KUKA KRL program: MyProgram_260().src

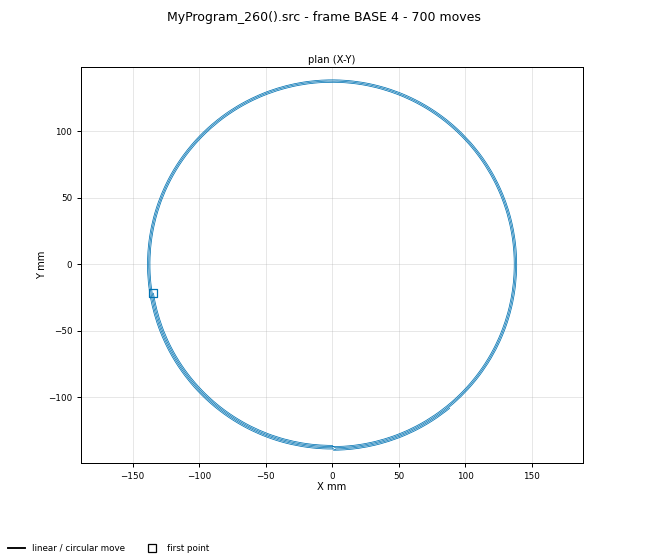
[picture p0: tool path of MyProgram_260().src in frame BASE 4, 700 of 700 moves have a stored position in this frame; points joined in program order, loops and branches not executed]
&ACCESS RVP
&REL 1
&PARAM TEMPLATE = C:\KRC\Roboter\Template\vorgabe
&PARAM EDITMASK = *
DEF MyProgram_260()
; ---- Setting reference (Base) ----
$BASE = BASE_DATA[4]

; --------------------------
; ---- Setting tool (TCP) ----
$TOOL = TOOL_DATA[3]
; --------------------------

$VEL.CP = VEL_APROX_PRINT
Startdeposition()
$VEL.CP = VEL_PRINT
LIN {X -134.3111,Y -21.6727,Z 167,A -169.5198,B 10.842,C 0.1896,E1 10.6856,E2 260.3687} C_DIS
LIN {X -133.7685,Y -24.8029,Z 167,A -167.9998,B 10.842,C 0.1897,E1 10.6864,E2 258.8275} C_DIS
LIN {X -133.0833,Y -28.2434,Z 167,A -166.7087,B 10.8418,C 0.1977,E1 10.6871,E2 257.5607} C_DIS
LIN {X -132.3432,Y -31.5283,Z 167,A -165.3421,B 10.8418,C 0.2028,E1 10.688,E2 256.2017} C_DIS
LIN {X -131.6516,Y -34.3082,Z 167,A -163.8428,B 10.8418,C 0.2002,E1 10.689,E2 254.6673} C_DIS
LIN {X -130.7834,Y -37.4821,Z 167,A -162.445,B 10.8418,C 0.2039,E1 10.6901,E2 253.2692} C_DIS
LIN {X -129.8475,Y -40.6068,Z 167,A -161.0737,B 10.8416,C 0.2077,E1 10.6912,E2 251.8994} C_DIS
LIN {X -128.6869,Y -44.1413,Z 167,A -159.7043,B 10.8415,C 0.216,E1 10.6924,E2 250.5557} C_DIS
LIN {X -127.68,Y -46.9788,Z 167,A -158.313,B 10.8415,C 0.217,E1 10.6937,E2 249.1502} C_DIS
LIN {X -126.4966,Y -50.0788,Z 167,A -156.7273,B 10.8415,C 0.2169,E1 10.6954,E2 247.5422} C_DIS
LIN {X -124.9844,Y -53.7359,Z 167,A -155.1801,B 10.8413,C 0.2238,E1 10.697,E2 246.0111} C_DIS
LIN {X -123.8203,Y -56.3713,Z 167,A -153.9567,B 10.8413,C 0.2268,E1 10.6984,E2 244.7874} C_DIS
LIN {X -122.3652,Y -59.4639,Z 167,A -152.3703,B 10.8413,C 0.2275,E1 10.7004,E2 243.1838} C_DIS
LIN {X -120.7964,Y -62.5886,Z 167,A -151.0422,B 10.8411,C 0.2342,E1 10.702,E2 241.8746} C_DIS
LIN {X -119.2164,Y -65.5493,Z 167,A -149.5746,B 10.8411,C 0.2367,E1 10.704,E2 240.4013} C_DIS
LIN {X -117.5118,Y -68.5582,Z 167,A -147.9691,B 10.8411,C 0.2372,E1 10.7063,E2 238.7782} C_DIS
LIN {X -115.1541,Y -72.4477,Z 167,A -146.0552,B 10.8409,C 0.2419,E1 10.7091,E2 236.8656} C_DIS
LIN {X -112.8943,Y -75.9219,Z 167,A -144.4013,B 10.8409,C 0.248,E1 10.7116,E2 235.2242} C_DIS
LIN {X -110.5948,Y -79.2332,Z 167,A -142.6335,B 10.8407,C 0.2505,E1 10.7145,E2 233.4487} C_DIS
LIN {X -108.3157,Y -82.3223,Z 167,A -141.0411,B 10.8407,C 0.2547,E1 10.7171,E2 231.8602} C_DIS
LIN {X -105.823,Y -85.502,Z 167,A -139.2465,B 10.8407,C 0.2565,E1 10.7203,E2 230.0548} C_DIS
LIN {X -103.3715,Y -88.4511,Z 167,A -137.6886,B 10.8405,C 0.2612,E1 10.7231,E2 228.5049} C_DIS
LIN {X -100.7123,Y -91.4665,Z 167,A -135.9235,B 10.8405,C 0.2633,E1 10.7264,E2 226.7314} C_DIS
LIN {X -97.6811,Y -94.6968,Z 167,A -134.0319,B 10.8404,C 0.2665,E1 10.73,E2 224.8374} C_DIS
LIN {X -94.874,Y -97.5096,Z 167,A -132.302,B 10.8404,C 0.2686,E1 10.7335,E2 223.1011} C_DIS
LIN {X -91.6335,Y -100.5608,Z 167,A -130.5474,B 10.8402,C 0.2748,E1 10.737,E2 221.3621} C_DIS
LIN {X -89.0111,Y -102.8893,Z 167,A -129.0545,B 10.8402,C 0.2771,E1 10.7402,E2 219.8677} C_DIS
LIN {X -86.4112,Y -105.0827,Z 167,A -127.5864,B 10.8401,C 0.2789,E1 10.7433,E2 218.3956} C_DIS
LIN {X -83.2289,Y -107.62,Z 167,A -125.805,B 10.8401,C 0.2804,E1 10.7473,E2 216.6062} C_DIS
LIN {X -80.1731,Y -109.916,Z 167,A -124.2299,B 10.8399,C 0.2838,E1 10.7508,E2 215.0358} C_DIS
LIN {X -77.3428,Y -111.9257,Z 167,A -122.6299,B 10.8399,C 0.2831,E1 10.7545,E2 213.4188} C_DIS
LIN {X -73.695,Y -114.3604,Z 167,A -120.8984,B 10.8399,C 0.2884,E1 10.7585,E2 211.7021} C_DIS
LIN {X -70.7703,Y -116.1931,Z 167,A -119.4359,B 10.8398,C 0.2903,E1 10.762,E2 210.2387} C_DIS
LIN {X -67.3111,Y -118.2299,Z 167,A -117.6848,B 10.8398,C 0.2913,E1 10.7662,E2 208.4801} C_DIS
LIN {X -63.9651,Y -120.0736,Z 167,A -116.1373,B 10.8397,C 0.2947,E1 10.77,E2 206.9405} C_DIS
LIN {X -60.9556,Y -121.6293,Z 167,A -114.5498,B 10.8397,C 0.2929,E1 10.774,E2 205.3328} C_DIS
LIN {X -57.4853,Y -123.3052,Z 167,A -113.1186,B 10.8395,C 0.299,E1 10.7776,E2 203.9257} C_DIS
LIN {X -54.7242,Y -124.557,Z 167,A -111.772,B 10.8395,C 0.2988,E1 10.781,E2 202.5703} C_DIS
LIN {X -51.6004,Y -125.8833,Z 167,A -110.3374,B 10.8395,C 0.3002,E1 10.7847,E2 201.1351} C_DIS
LIN {X -48.507,Y -127.1076,Z 167,A -108.9314,B 10.8395,C 0.3014,E1 10.7884,E2 199.7283} C_DIS
LIN {X -45.354,Y -128.2665,Z 167,A -107.4225,B 10.8395,C 0.3005,E1 10.7924,E2 198.2074} C_DIS
LIN {X -42.1439,Y -129.3565,Z 167,A -106.0814,B 10.8395,C 0.3036,E1 10.7959,E2 196.8771} C_DIS
LIN {X -39.0213,Y -130.3327,Z 167,A -104.7004,B 10.8394,C 0.3045,E1 10.7996,E2 195.4955} C_DIS
LIN {X -35.848,Y -131.241,Z 167,A -103.3079,B 10.8394,C 0.3054,E1 10.8033,E2 194.1024} C_DIS
LIN {X -32.179,Y -132.1863,Z 167,A -101.6912,B 10.8394,C 0.3058,E1 10.8077,E2 192.4826} C_DIS
LIN {X -29.0348,Y -132.9124,Z 167,A -100.3891,B 10.8393,C 0.3079,E1 10.8112,E2 191.1873} C_DIS
LIN {X -26.3362,Y -133.4754,Z 167,A -99.1709,B 10.8393,C 0.3071,E1 10.8146,E2 189.9617} C_DIS
LIN {X -23.131,Y -134.0678,Z 167,A -97.833,B 10.8393,C 0.3084,E1 10.8183,E2 188.6278} C_DIS
LIN {X -19.4524,Y -134.6488,Z 167,A -96.2396,B 10.8393,C 0.3084,E1 10.8227,E2 187.0307} C_DIS
LIN {X -15.3344,Y -135.1819,Z 167,A -94.4826,B 10.8393,C 0.3085,E1 10.8276,E2 185.2721} C_DIS
LIN {X -12.2246,Y -135.4985,Z 167,A -93.1676,B 10.8393,C 0.3088,E1 10.8312,E2 183.9568} C_DIS
LIN {X -9.0884,Y -135.7447,Z 167,A -91.8792,B 10.8393,C 0.3097,E1 10.8348,E2 182.6725} C_DIS
LIN {X -6.0197,Y -135.9153,Z 167,A -90.4241,B 10.8393,C 0.3059,E1 10.8389,E2 181.1965} C_DIS
LIN {X -3.0197,Y -136.0153,Z 167,A -89.3083,B 10.8393,C 0.3094,E1 10.842,E2 180.0989} C_DIS
LIN {X 0.0448,Y -136.0486,Z 167,A -88.0199,B 10.8393,C 0.3093,E1 10.8456,E2 178.8102} C_DIS
LIN {X 0.0448,Y -136.0486,Z 167,A -88.0199,B 10.8393,C 0.3093,E1 10.8456,E2 178.8102} C_DIS
Enddeposition()
LIN {X 0.9674,Y -136.9518,Z 167,A -88.835,B 10.7499,C 0.3477,E1 10.7545,E2 179.837} C_DIS
Startdeposition()
$VEL.CP = VEL_PRINT
LIN {X -4.7131,Y -136.8825,Z 167,A -90.5763,B 10.7503,C 0.333,E1 10.7499,E2 181.5002} C_DIS
LIN {X -10.8547,Y -136.533,Z 167,A -93.0554,B 10.7503,C 0.3307,E1 10.743,E2 183.9685} C_DIS
LIN {X -17.1623,Y -135.8841,Z 167,A -95.8644,B 10.7503,C 0.3338,E1 10.7351,E2 186.7983} C_DIS
LIN {X -20.236,Y -135.4608,Z 167,A -97.0548,B 10.7503,C 0.331,E1 10.7319,E2 187.9756} C_DIS
LIN {X -22.5354,Y -135.0954,Z 167,A -98.3975,B 10.7501,C 0.3391,E1 10.728,E2 189.3648} C_DIS
LIN {X -26.0699,Y -134.4585,Z 167,A -99.6085,B 10.7504,C 0.3318,E1 10.7248,E2 190.5397} C_DIS
LIN {X -30.2799,Y -133.573,Z 167,A -101.349,B 10.7504,C 0.3295,E1 10.7201,E2 192.2732} C_DIS
LIN {X -33.8041,Y -132.7248,Z 167,A -102.7917,B 10.7504,C 0.327,E1 10.7162,E2 193.707} C_DIS
LIN {X -36.2381,Y -132.0826,Z 167,A -103.8721,B 10.7504,C 0.327,E1 10.7133,E2 194.791} C_DIS
LIN {X -40.0727,Y -130.9684,Z 167,A -105.5983,B 10.7504,C 0.327,E1 10.7086,E2 196.5245} C_DIS
LIN {X -43.2695,Y -129.9473,Z 167,A -106.9315,B 10.7506,C 0.3243,E1 10.7051,E2 197.8489} C_DIS
LIN {X -45.7774,Y -129.0871,Z 167,A -108.0875,B 10.7506,C 0.3245,E1 10.702,E2 199.0111} C_DIS
LIN {X -49.2408,Y -127.8047,Z 167,A -109.7273,B 10.7506,C 0.3252,E1 10.6977,E2 200.6629} C_DIS
LIN {X -53.1385,Y -126.2338,Z 167,A -112.0436,B 10.7502,C 0.3357,E1 10.6916,E2 203.0489} C_DIS
LIN {X -57.5437,Y -124.2869,Z 167,A -113.504,B 10.7507,C 0.3213,E1 10.6881,E2 204.4402} C_DIS
LIN {X -61.4514,Y -122.4043,Z 167,A -115.2744,B 10.7507,C 0.3182,E1 10.6836,E2 206.2051} C_DIS
LIN {X -64.9538,Y -120.5822,Z 167,A -117.0541,B 10.7507,C 0.3189,E1 10.6792,E2 208.0007} C_DIS
LIN {X -68.8615,Y -118.3944,Z 167,A -118.9424,B 10.7508,C 0.3167,E1 10.6746,E2 209.8907} C_DIS
LIN {X -72.4707,Y -116.2199,Z 167,A -120.6707,B 10.7508,C 0.3135,E1 10.6705,E2 211.6145} C_DIS
LIN {X -76.087,Y -113.8851,Z 167,A -122.5284,B 10.7509,C 0.312,E1 10.6661,E2 213.479} C_DIS
LIN {X -79.7805,Y -111.329,Z 167,A -124.399,B 10.751,C 0.3088,E1 10.6619,E2 215.3482} C_DIS
LIN {X -83.3183,Y -108.7066,Z 167,A -126.2772,B 10.751,C 0.3065,E1 10.6577,E2 217.2305} C_DIS
LIN {X -86.7761,Y -105.9668,Z 167,A -128.1009,B 10.7512,C 0.3029,E1 10.6537,E2 219.051} C_DIS
LIN {X -89.8766,Y -103.3504,Z 167,A -129.9044,B 10.7512,C 0.302,E1 10.6499,E2 220.8671} C_DIS
LIN {X -93.4491,Y -100.1316,Z 167,A -131.8374,B 10.7514,C 0.2966,E1 10.6459,E2 222.7897} C_DIS
LIN {X -96.4913,Y -97.2033,Z 167,A -133.6849,B 10.7514,C 0.2948,E1 10.6422,E2 224.6466} C_DIS
LIN {X -99.7788,Y -93.8258,Z 167,A -135.5661,B 10.7516,C 0.2889,E1 10.6386,E2 226.5158} C_DIS
LIN {X -102.2245,Y -91.1553,Z 167,A -137.0213,B 10.7516,C 0.2845,E1 10.6359,E2 227.9628} C_DIS
LIN {X -104.9392,Y -88.0159,Z 167,A -138.9347,B 10.7516,C 0.2845,E1 10.6323,E2 229.8975} C_DIS
LIN {X -107.5627,Y -84.7901,Z 167,A -140.6791,B 10.7518,C 0.2807,E1 10.6293,E2 231.6416} C_DIS
LIN {X -110.1564,Y -81.3926,Z 167,A -142.5582,B 10.7518,C 0.2785,E1 10.6261,E2 233.5311} C_DIS
LIN {X -112.8424,Y -77.6251,Z 167,A -144.4788,B 10.752,C 0.2737,E1 10.6231,E2 235.4487} C_DIS
LIN {X -115.3626,Y -73.8276,Z 167,A -146.3667,B 10.752,C 0.2687,E1 10.6202,E2 237.3331} C_DIS
LIN {X -117.4555,Y -70.4514,Z 167,A -148.0697,B 10.7522,C 0.2655,E1 10.6177,E2 239.0402} C_DIS
LIN {X -119.535,Y -66.8619,Z 167,A -149.7167,B 10.7523,C 0.2594,E1 10.6154,E2 240.6752} C_DIS
LIN {X -121.1719,Y -63.8429,Z 167,A -151.1675,B 10.7524,C 0.256,E1 10.6135,E2 242.1266} C_DIS
LIN {X -122.6969,Y -60.8609,Z 167,A -152.4431,B 10.7525,C 0.2498,E1 10.6119,E2 243.3856} C_DIS
LIN {X -124.2372,Y -57.6513,Z 167,A -154.2089,B 10.7525,C 0.2516,E1 10.6098,E2 245.1847} C_DIS
LIN {X -125.8288,Y -54.0898,Z 167,A -155.7963,B 10.7526,C 0.2464,E1 10.608,E2 246.7653} C_DIS
LIN {X -127.3195,Y -50.4864,Z 167,A -157.5839,B 10.7526,C 0.2452,E1 10.6061,E2 248.5711} C_DIS
LIN {X -128.6089,Y -47.1037,Z 167,A -159.3622,B 10.7526,C 0.2464,E1 10.6044,E2 250.3806} C_DIS
LIN {X -129.8916,Y -43.4367,Z 167,A -160.5546,B 10.7529,C 0.2332,E1 10.6034,E2 251.5184} C_DIS
LIN {X -131.8065,Y -37.2253,Z 167,A -163.3987,B 10.753,C 0.2282,E1 10.6011,E2 254.3757} C_DIS
LIN {X -132.6261,Y -34.1929,Z 167,A -164.7615,B 10.753,C 0.2255,E1 10.6001,E2 255.7434} C_DIS
LIN {X -133.5136,Y -30.54,Z 167,A -166.2733,B 10.7532,C 0.2198,E1 10.5991,E2 257.2463} C_DIS
LIN {X -134.1919,Y -27.4069,Z 167,A -167.6224,B 10.7532,C 0.2161,E1 10.5983,E2 258.5952} C_DIS
LIN {X -134.7947,Y -24.2694,Z 167,A -168.8911,B 10.7534,C 0.2109,E1 10.5977,E2 259.8543} C_DIS
LIN {X -135.2987,Y -21.2831,Z 167,A -170.3335,B 10.7534,C 0.2109,E1 10.597,E2 261.3171} C_DIS
LIN {X -135.796,Y -17.8342,Z 167,A -171.7984,B 10.7534,C 0.2067,E1 10.5965,E2 262.7815} C_DIS
LIN {X -136.2655,Y -13.8156,Z 167,A -173.6079,B 10.7534,C 0.2042,E1 10.5959,E2 264.6038} C_DIS
LIN {X -136.5962,Y -10.006,Z 167,A -175.108,B 10.7536,C 0.1975,E1 10.5956,E2 266.0901} C_DIS
LIN {X -136.7995,Y -6.6765,Z 167,A -176.6098,B 10.7536,C 0.1955,E1 10.5954,E2 267.6036} C_DIS
LIN {X -136.928,Y -3.1345,Z 167,A -178.1573,B 10.7537,C 0.1925,E1 10.5952,E2 269.1575} C_DIS
LIN {X -136.955,Y 1.577,Z 167,A 179.9462,B 10.7538,C 0.1852,E1 10.5952,E2 271.0429} C_DIS
LIN {X -136.8559,Y 5.397,Z 167,A 178.2914,B 10.7538,C 0.1817,E1 10.5954,E2 272.703} C_DIS
LIN {X -136.6019,Y 9.9282,Z 167,A 176.5847,B 10.754,C 0.1723,E1 10.5957,E2 274.3841} C_DIS
LIN {X -136.4146,Y 12.2532,Z 167,A 175.2503,B 10.754,C 0.1765,E1 10.596,E2 275.7615} C_DIS
LIN {X -135.9101,Y 16.9595,Z 167,A 173.4502,B 10.7541,C 0.1672,E1 10.5966,E2 277.5374} C_DIS
LIN {X -135.3658,Y 20.8497,Z 167,A 171.7505,B 10.7541,C 0.1635,E1 10.5973,E2 279.2423} C_DIS
LIN {X -134.7404,Y 24.5729,Z 167,A 170.1227,B 10.7542,C 0.1599,E1 10.598,E2 280.8743} C_DIS
LIN {X -133.9418,Y 28.6053,Z 167,A 168.3826,B 10.7543,C 0.1553,E1 10.599,E2 282.615} C_DIS
LIN {X -133.1867,Y 31.936,Z 167,A 167.062,B 10.7543,C 0.1491,E1 10.5998,E2 283.9207} C_DIS
LIN {X -132.5445,Y 34.5131,Z 167,A 165.6782,B 10.7543,C 0.1513,E1 10.6008,E2 285.3368} C_DIS
LIN {X -131.191,Y 39.3454,Z 167,A 163.608,B 10.7544,C 0.1448,E1 10.6024,E2 287.4011} C_DIS
LIN {X -129.0397,Y 45.9089,Z 167,A 160.7075,B 10.7546,C 0.1369,E1 10.605,E2 290.2997} C_DIS
LIN {X -128.0145,Y 48.696,Z 167,A 159.3753,B 10.7546,C 0.1353,E1 10.6063,E2 291.6415} C_DIS
LIN {X -126.5439,Y 52.3959,Z 167,A 158.002,B 10.7546,C 0.1249,E1 10.6077,E2 292.9773} C_DIS
LIN {X -125.519,Y 54.8064,Z 167,A 156.5707,B 10.7546,C 0.1286,E1 10.6094,E2 294.4483} C_DIS
LIN {X -123.9382,Y 58.2967,Z 167,A 154.9657,B 10.7547,C 0.1244,E1 10.6112,E2 296.0518} C_DIS
LIN {X -121.5401,Y 63.1415,Z 167,A 152.733,B 10.7547,C 0.1178,E1 10.614,E2 298.2785} C_DIS
LIN {X -119.3595,Y 67.1741,Z 167,A 150.8289,B 10.7548,C 0.1125,E1 10.6166,E2 300.1788} C_DIS
LIN {X -117.3366,Y 70.6488,Z 167,A 149.0969,B 10.7548,C 0.1092,E1 10.6191,E2 301.915} C_DIS
LIN {X -115.065,Y 74.2914,Z 167,A 147.2245,B 10.7548,C 0.1063,E1 10.6219,E2 303.7948} C_DIS
LIN {X -112.5356,Y 78.0693,Z 167,A 145.3511,B 10.7549,C 0.101,E1 10.6248,E2 305.6625} C_DIS
LIN {X -110.0057,Y 81.5957,Z 167,A 143.4661,B 10.7549,C 0.0981,E1 10.6279,E2 307.554} C_DIS
LIN {X -107.3781,Y 85.0241,Z 167,A 141.7213,B 10.755,C 0.0926,E1 10.6309,E2 309.2893} C_DIS
LIN {X -105.0064,Y 87.9358,Z 167,A 140.2729,B 10.755,C 0.0864,E1 10.6334,E2 310.7211} C_DIS
LIN {X -103.2358,Y 90.0079,Z 167,A 138.6961,B 10.755,C 0.0927,E1 10.6364,E2 312.3496} C_DIS
LIN {X -100.9472,Y 92.5675,Z 167,A 137.4613,B 10.755,C 0.0855,E1 10.6387,E2 313.5585} C_DIS
LIN {X -97.9081,Y 95.7762,Z 167,A 135.5774,B 10.7551,C 0.0822,E1 10.6424,E2 315.4447} C_DIS
LIN {X -94.8928,Y 98.765,Z 167,A 133.2307,B 10.7551,C 0.0902,E1 10.6472,E2 317.8583} C_DIS
LIN {X -91.0041,Y 102.3594,Z 167,A 131.6541,B 10.7551,C 0.0727,E1 10.6503,E2 319.3558} C_DIS
LIN {X -84.9127,Y 107.4661,Z 167,A 127.8282,B 10.7551,C 0.0767,E1 10.6587,E2 323.2389} C_DIS
LIN {X -81.4986,Y 110.078,Z 167,A 126.4245,B 10.7552,C 0.0653,E1 10.6617,E2 324.5931} C_DIS
LIN {X -77.8583,Y 112.6824,Z 167,A 124.7002,B 10.7552,C 0.059,E1 10.6656,E2 326.2977} C_DIS
LIN {X -73.6068,Y 115.504,Z 167,A 122.3089,B 10.7552,C 0.0608,E1 10.6713,E2 328.7182} C_DIS
LIN {X -69.7893,Y 117.8502,Z 167,A 120.5095,B 10.7552,C 0.0563,E1 10.6755,E2 330.5068} C_DIS
LIN {X -66.3051,Y 119.8444,Z 167,A 118.8548,B 10.7552,C 0.0533,E1 10.6796,E2 332.1569} C_DIS
LIN {X -62.6236,Y 121.8076,Z 167,A 117.0539,B 10.7552,C 0.052,E1 10.684,E2 333.963} C_DIS
LIN {X -59.2444,Y 123.4855,Z 167,A 115.5288,B 10.7553,C 0.0488,E1 10.6878,E2 335.4802} C_DIS
LIN {X -56.047,Y 124.969,Z 167,A 114.1459,B 10.7553,C 0.045,E1 10.6913,E2 336.8508} C_DIS
LIN {X -53.5557,Y 126.0595,Z 167,A 112.912,B 10.7553,C 0.0457,E1 10.6945,E2 338.0955} C_DIS
LIN {X -49.0971,Y 127.8606,Z 167,A 110.7792,B 10.7553,C 0.046,E1 10.7001,E2 340.2413} C_DIS
LIN {X -41.6451,Y 130.4769,Z 167,A 107.5869,B 10.7553,C 0.0403,E1 10.7085,E2 343.4175} C_DIS
LIN {X -38.4851,Y 131.4437,Z 167,A 106.2648,B 10.7553,C 0.0378,E1 10.712,E2 344.7314} C_DIS
LIN {X -35.3859,Y 132.3118,Z 167,A 104.8302,B 10.7553,C 0.0386,E1 10.7159,E2 346.1757} C_DIS
LIN {X -32.1849,Y 133.1267,Z 167,A 103.5357,B 10.7553,C 0.0356,E1 10.7193,E2 347.4586} C_DIS
LIN {X -29.1697,Y 133.82,Z 167,A 102.0742,B 10.7553,C 0.0384,E1 10.7234,E2 348.9396} C_DIS
LIN {X -25.0151,Y 134.6601,Z 167,A 100.3769,B 10.7553,C 0.0357,E1 10.728,E2 350.6266} C_DIS
LIN {X -21.0529,Y 135.3344,Z 167,A 98.7868,B 10.7553,C 0.0328,E1 10.7324,E2 352.2045} C_DIS
LIN {X -18.626,Y 135.6917,Z 167,A 97.4583,B 10.7553,C 0.0391,E1 10.7361,E2 353.5692} C_DIS
LIN {X -13.6092,Y 136.2853,Z 167,A 95.4594,B 10.7553,C 0.0357,E1 10.7416,E2 355.5529} C_DIS
LIN {X -10.0887,Y 136.5901,Z 167,A 94.0503,B 10.7553,C 0.0337,E1 10.7455,E2 356.9528} C_DIS
LIN {X -6.1839,Y 136.8243,Z 167,A 92.1888,B 10.7553,C 0.0385,E1 10.7508,E2 358.8409} C_DIS
LIN {X 1.1285,Y 136.9581,Z 167,A 89.2887,B 10.7553,C 0.0347,E1 10.7588,E2 361.7201} C_DIS
LIN {X 4.4358,Y 136.8919,Z 167,A 87.2804,B 10.7553,C 0.0489,E1 10.7647,E2 363.8033} C_DIS
LIN {X 9.7416,Y 136.6155,Z 167,A 85.5485,B 10.7553,C 0.0381,E1 10.7693,E2 365.4752} C_DIS
LIN {X 14.5162,Y 136.1908,Z 167,A 83.7262,B 10.7553,C 0.0343,E1 10.7743,E2 367.2745} C_DIS
LIN {X 18.4906,Y 135.71,Z 167,A 82.0233,B 10.7553,C 0.0356,E1 10.779,E2 368.9804} C_DIS
LIN {X 22.965,Y 135.0237,Z 167,A 80.0536,B 10.7553,C 0.0381,E1 10.7845,E2 370.9587} C_DIS
LIN {X 27.1076,Y 134.2528,Z 167,A 78.4933,B 10.7553,C 0.0343,E1 10.7887,E2 372.4939} C_DIS
LIN {X 30.2962,Y 133.5693,Z 167,A 77.0576,B 10.7553,C 0.0368,E1 10.7926,E2 373.938} C_DIS
LIN {X 33.1964,Y 132.879,Z 167,A 75.6644,B 10.7553,C 0.041,E1 10.7965,E2 375.3487} C_DIS
LIN {X 37.4201,Y 131.752,Z 167,A 73.901,B 10.7553,C 0.0408,E1 10.8012,E2 377.1039} C_DIS
LIN {X 41.3615,Y 130.5675,Z 167,A 72.3809,B 10.7553,C 0.0374,E1 10.8052,E2 378.5991} C_DIS
LIN {X 43.9327,Y 129.7264,Z 167,A 71.0388,B 10.7553,C 0.0435,E1 10.8088,E2 379.9668} C_DIS
LIN {X 47.8009,Y 128.3498,Z 167,A 69.5492,B 10.7553,C 0.0396,E1 10.8126,E2 381.4283} C_DIS
LIN {X 49.8612,Y 127.5635,Z 167,A 68.3622,B 10.7553,C 0.0469,E1 10.8158,E2 382.6476} C_DIS
LIN {X 53.535,Y 126.068,Z 167,A 66.8109,B 10.7553,C 0.0461,E1 10.8198,E2 384.1857} C_DIS
LIN {X 56.9866,Y 124.5445,Z 167,A 65.255,B 10.7553,C 0.0474,E1 10.8237,E2 385.7389} C_DIS
LIN {X 59.7901,Y 123.2248,Z 167,A 63.843,B 10.7553,C 0.0518,E1 10.8273,E2 387.1651} C_DIS
LIN {X 63.4519,Y 121.3772,Z 167,A 62.2684,B 10.7553,C 0.0506,E1 10.8312,E2 388.7224} C_DIS
LIN {X 67.4473,Y 119.206,Z 167,A 60.3552,B 10.7553,C 0.0535,E1 10.8359,E2 390.6373} C_DIS
LIN {X 70.9231,Y 117.1707,Z 167,A 58.656,B 10.7553,C 0.0563,E1 10.84,E2 392.3384} C_DIS
LIN {X 74.4855,Y 114.939,Z 167,A 56.9297,B 10.7553,C 0.0582,E1 10.844,E2 394.0611} C_DIS
LIN {X 77.9554,Y 112.6149,Z 167,A 55.1446,B 10.7553,C 0.0619,E1 10.8481,E2 395.8511} C_DIS
LIN {X 81.6123,Y 109.9933,Z 167,A 53.3141,B 10.7553,C 0.0638,E1 10.8523,E2 397.6756} C_DIS
LIN {X 84.8356,Y 107.527,Z 167,A 51.5987,B 10.7553,C 0.0673,E1 10.8561,E2 399.3937} C_DIS
LIN {X 88.0435,Y 104.9161,Z 167,A 49.891,B 10.7552,C 0.0699,E1 10.8597,E2 401.0991} C_DIS
LIN {X 91.6118,Y 101.8157,Z 167,A 47.958,B 10.7552,C 0.0725,E1 10.8638,E2 403.0274} C_DIS
LIN {X 94.0854,Y 99.5339,Z 167,A 46.5202,B 10.7552,C 0.076,E1 10.8667,E2 404.4693} C_DIS
LIN {X 97.4738,Y 96.2191,Z 167,A 44.6018,B 10.7552,C 0.0784,E1 10.8705,E2 406.3806} C_DIS
LIN {X 99.8919,Y 93.7059,Z 167,A 42.7946,B 10.755,C 0.0902,E1 10.874,E2 408.231} C_DIS
LIN {X 102.631,Y 90.6968,Z 167,A 41.4667,B 10.755,C 0.0845,E1 10.8764,E2 409.5139} C_DIS
LIN {X 105.1386,Y 87.7784,Z 167,A 39.9317,B 10.755,C 0.0861,E1 10.8792,E2 411.0405} C_DIS
LIN {X 107.6593,Y 84.6671,Z 167,A 38.1663,B 10.755,C 0.0922,E1 10.8823,E2 412.8178} C_DIS
LIN {X 110.5884,Y 80.8045,Z 167,A 36.1879,B 10.755,C 0.0956,E1 10.8855,E2 414.7912} C_DIS
LIN {X 112.8658,Y 77.591,Z 167,A 34.6046,B 10.755,C 0.0979,E1 10.8881,E2 416.3675} C_DIS
LIN {X 115.2515,Y 74.0012,Z 167,A 32.7816,B 10.755,C 0.1028,E1 10.8909,E2 418.194} C_DIS
LIN {X 117.597,Y 70.214,Z 167,A 30.9375,B 10.7549,C 0.1069,E1 10.8935,E2 420.0369} C_DIS
LIN {X 119.0686,Y 67.6888,Z 167,A 29.611,B 10.7549,C 0.1126,E1 10.8954,E2 421.377} C_DIS
LIN {X 121.6295,Y 62.9714,Z 167,A 27.483,B 10.7549,C 0.1153,E1 10.8982,E2 423.4921} C_DIS
LIN {X 123.1787,Y 59.8844,Z 167,A 25.9587,B 10.7547,C 0.1212,E1 10.9001,E2 425.0272} C_DIS
LIN {X 124.8815,Y 56.2428,Z 167,A 24.4554,B 10.7547,C 0.121,E1 10.9018,E2 426.5097} C_DIS
LIN {X 126.1896,Y 53.2442,Z 167,A 23.3047,B 10.7547,C 0.119,E1 10.903,E2 427.6343} C_DIS
LIN {X 127.5141,Y 49.9884,Z 167,A 21.8935,B 10.7547,C 0.1214,E1 10.9045,E2 429.0393} C_DIS
LIN {X 129.1296,Y 45.6595,Z 167,A 19.6691,B 10.7546,C 0.1343,E1 10.9067,E2 431.3016} C_DIS
LIN {X 130.4263,Y 41.8037,Z 167,A 18.0967,B 10.7546,C 0.1356,E1 10.908,E2 432.8592} C_DIS
LIN {X 131.5778,Y 38.027,Z 167,A 16.3697,B 10.7545,C 0.1422,E1 10.9094,E2 434.597} C_DIS
LIN {X 132.6948,Y 33.922,Z 167,A 14.7868,B 10.7545,C 0.142,E1 10.9105,E2 436.157} C_DIS
LIN {X 133.412,Y 30.9847,Z 167,A 13.622,B 10.7545,C 0.143,E1 10.9112,E2 437.3105} C_DIS
LIN {X 134.3004,Y 26.8734,Z 167,A 11.7105,B 10.7543,C 0.152,E1 10.9124,E2 439.2425} C_DIS
LIN {X 135.0602,Y 22.7458,Z 167,A 10.2026,B 10.7543,C 0.1506,E1 10.9131,E2 440.7211} C_DIS
LIN {X 135.582,Y 19.3937,Z 167,A 8.5858,B 10.7543,C 0.1599,E1 10.9138,E2 442.3639} C_DIS
LIN {X 136.052,Y 15.77,Z 167,A 6.8305,B 10.7541,C 0.1703,E1 10.9144,E2 444.1488} C_DIS
LIN {X 136.4031,Y 12.3826,Z 167,A 5.7294,B 10.7541,C 0.1659,E1 10.9146,E2 445.2112} C_DIS
LIN {X 136.6438,Y 9.3533,Z 167,A 3.9572,B 10.7539,C 0.1828,E1 10.915,E2 447.0468} C_DIS
LIN {X 136.8746,Y 4.9172,Z 167,A 2.8097,B 10.7541,C 0.1696,E1 10.9151,E2 448.1078} C_DIS
LIN {X 136.9587,Y 1.0634,Z 167,A 0.7255,B 10.7538,C 0.1867,E1 10.9152,E2 450.2525} C_DIS
LIN {X 136.9424,Y -2.334,Z 167,A -0.3407,B 10.7538,C 0.1815,E1 10.9152,E2 451.2759} C_DIS
LIN {X 136.7563,Y -7.5372,Z 167,A -2.5181,B 10.7538,C 0.1879,E1 10.9149,E2 453.4555} C_DIS
LIN {X 136.5174,Y -11.0398,Z 167,A -3.8497,B 10.7538,C 0.1886,E1 10.9147,E2 454.7715} C_DIS
LIN {X 136.2562,Y -13.9057,Z 167,A -5.2303,B 10.7536,C 0.1968,E1 10.9143,E2 456.1755} C_DIS
LIN {X 135.8765,Y -17.2199,Z 167,A -6.4909,B 10.7536,C 0.1973,E1 10.9139,E2 457.4208} C_DIS
LIN {X 135.4655,Y -20.2056,Z 167,A -7.7273,B 10.7536,C 0.2004,E1 10.9134,E2 458.6555} C_DIS
LIN {X 134.6213,Y -25.2178,Z 167,A -9.9847,B 10.7534,C 0.21,E1 10.9123,E2 460.9316} C_DIS
LIN {X 133.7447,Y -29.5183,Z 167,A -11.6364,B 10.7534,C 0.2105,E1 10.9113,E2 462.5622} C_DIS
LIN {X 133.1651,Y -32.0255,Z 167,A -12.7324,B 10.7534,C 0.2141,E1 10.9106,E2 463.6618} C_DIS
LIN {X 132.0957,Y -36.1911,Z 167,A -14.5986,B 10.7532,C 0.221,E1 10.9093,E2 465.5385} C_DIS
LIN {X 131.0307,Y -39.8691,Z 167,A -16.0396,B 10.7532,C 0.2213,E1 10.9082,E2 466.961} C_DIS
LIN {X 130.0638,Y -42.9196,Z 167,A -17.2899,B 10.7532,C 0.2228,E1 10.9071,E2 468.2017} C_DIS
LIN {X 128.9501,Y -46.1575,Z 167,A -18.6852,B 10.7531,C 0.2258,E1 10.9058,E2 469.594} C_DIS
LIN {X 128.1703,Y -48.2802,Z 167,A -20.104,B 10.7527,C 0.2409,E1 10.9044,E2 471.0732} C_DIS
LIN {X 126.8356,Y -51.6868,Z 167,A -21.3201,B 10.7528,C 0.2368,E1 10.9031,E2 472.2517} C_DIS
LIN {X 125.2802,Y -55.3513,Z 167,A -23.1251,B 10.7527,C 0.2451,E1 10.9011,E2 474.076} C_DIS
LIN {X 123.0411,Y -60.1633,Z 167,A -25.3906,B 10.7525,C 0.2522,E1 10.8984,E2 476.3497} C_DIS
LIN {X 121.5475,Y -63.1276,Z 167,A -26.5616,B 10.7525,C 0.2502,E1 10.8969,E2 477.4949} C_DIS
LIN {X 119.3203,Y -67.2439,Z 167,A -28.4965,B 10.7525,C 0.2548,E1 10.8943,E2 479.4292} C_DIS
LIN {X 117.2033,Y -70.8691,Z 167,A -30.2109,B 10.7523,C 0.2582,E1 10.8918,E2 481.1403} C_DIS
LIN {X 114.8613,Y -74.6052,Z 167,A -31.9966,B 10.7523,C 0.2614,E1 10.8892,E2 482.9206} C_DIS
LIN {X 112.7797,Y -77.7165,Z 167,A -33.5243,B 10.7523,C 0.2643,E1 10.8868,E2 484.4453} C_DIS
LIN {X 110.6095,Y -80.7757,Z 167,A -35.0817,B 10.7521,C 0.2678,E1 10.8842,E2 486.003} C_DIS
LIN {X 107.9411,Y -84.3084,Z 167,A -36.719,B 10.7521,C 0.2667,E1 10.8815,E2 487.6152} C_DIS
LIN {X 104.2888,Y -88.7858,Z 167,A -39.8326,B 10.7515,C 0.2903,E1 10.8758,E2 490.819} C_DIS
LIN {X 101.1751,Y -92.319,Z 167,A -41.3986,B 10.7517,C 0.2844,E1 10.873,E2 492.3366} C_DIS
LIN {X 98.0589,Y -95.6224,Z 167,A -43.1823,B 10.7517,C 0.2856,E1 10.8695,E2 494.1077} C_DIS
LIN {X 95.2871,Y -98.384,Z 167,A -44.77,B 10.7517,C 0.2878,E1 10.8664,E2 495.6909} C_DIS
LIN {X 92.3309,Y -101.1642,Z 167,A -46.282,B 10.7517,C 0.2866,E1 10.8633,E2 497.1812} C_DIS
LIN {X 89.7116,Y -103.4943,Z 167,A -48.0012,B 10.7514,C 0.296,E1 10.8597,E2 498.9339} C_DIS
LIN {X 86.4047,Y -106.2704,Z 167,A -49.6966,B 10.7514,C 0.2967,E1 10.856,E2 500.6171} C_DIS
LIN {X 83.364,Y -108.6716,Z 167,A -51.312,B 10.7513,C 0.2997,E1 10.8525,E2 502.2335} C_DIS
LIN {X 80.8037,Y -110.589,Z 167,A -52.735,B 10.7512,C 0.3043,E1 10.8492,E2 503.6685} C_DIS
LIN {X 77.023,Y -113.2546,Z 167,A -54.6081,B 10.7512,C 0.3062,E1 10.845,E2 505.5357} C_DIS
LIN {X 70.6944,Y -117.309,Z 167,A -57.726,B 10.751,C 0.3108,E1 10.8376,E2 508.6533} C_DIS
LIN {X 66.9669,Y -119.476,Z 167,A -59.4674,B 10.751,C 0.312,E1 10.8334,E2 510.3885} C_DIS
LIN {X 63.2028,Y -121.5079,Z 167,A -61.4097,B 10.7508,C 0.3185,E1 10.8285,E2 512.3517} C_DIS
LIN {X 57.7125,Y -124.2088,Z 167,A -63.6946,B 10.7508,C 0.3152,E1 10.8229,E2 514.6041} C_DIS
LIN {X 55.0689,Y -125.4055,Z 167,A -64.919,B 10.7508,C 0.3171,E1 10.8197,E2 515.8309} C_DIS
LIN {X 51.6598,Y -126.8465,Z 167,A -66.417,B 10.7508,C 0.3177,E1 10.8159,E2 517.3238} C_DIS
LIN {X 48.3319,Y -128.1509,Z 167,A -67.9481,B 10.7507,C 0.3204,E1 10.8119,E2 518.8606} C_DIS
LIN {X 45.1423,Y -129.3089,Z 167,A -69.3861,B 10.7507,C 0.3224,E1 10.8081,E2 520.3021} C_DIS
LIN {X 41.9049,Y -130.394,Z 167,A -70.7108,B 10.7507,C 0.3213,E1 10.8046,E2 521.6148} C_DIS
LIN {X 39.3203,Y -131.1986,Z 167,A -72.1089,B 10.7504,C 0.329,E1 10.8008,E2 523.0473} C_DIS
LIN {X 35.4625,Y -132.2914,Z 167,A -73.4514,B 10.7506,C 0.3223,E1 10.7973,E2 524.3488} C_DIS
LIN {X 32.7466,Y -132.9913,Z 167,A -74.7041,B 10.7506,C 0.3252,E1 10.7939,E2 525.6124} C_DIS
LIN {X 29.1087,Y -133.8331,Z 167,A -76.2064,B 10.7506,C 0.325,E1 10.7898,E2 527.1082} C_DIS
LIN {X 24.6952,Y -134.7185,Z 167,A -78.2498,B 10.7504,C 0.3302,E1 10.7841,E2 529.1731} C_DIS
LIN {X 21.0542,Y -135.3342,Z 167,A -79.8674,B 10.7504,C 0.3328,E1 10.7796,E2 530.8009} C_DIS
LIN {X 16.573,Y -135.9562,Z 167,A -81.6602,B 10.7504,C 0.3314,E1 10.7747,E2 532.5823} C_DIS
LIN {X 13.1235,Y -136.332,Z 167,A -83.6483,B 10.7499,C 0.3448,E1 10.769,E2 534.6385} C_DIS
LIN {X 8.3808,Y -136.7055,Z 167,A -85.9323,B 10.7497,C 0.3523,E1 10.7625,E2 536.9602} C_DIS
LIN {X 2.0214,Y -136.9476,Z 167,A -87.4405,B 10.7505,C 0.3257,E1 10.7587,E2 538.325} C_DIS
LIN {X 0.9674,Y -136.9518,Z 167,A -88.8328,B 10.7498,C 0.3481,E1 10.7545,E2 539.837} C_DIS
Enddeposition()
LIN {X 0.9674,Y -136.9518,Z 167,A -88.8328,B 10.7498,C 0.3481,E1 10.7545,E2 539.837} C_DIS
Startdeposition()
$VEL.CP = VEL_PRINT
LIN {X 2.6157,Y -137.8534,Z 167,A -86.496,B 10.6618,C 0.3189,E1 10.6726,E2 537.3517} C_DIS
LIN {X 6.0526,Y -137.7466,Z 167,A -85.2714,B 10.6618,C 0.3235,E1 10.6759,E2 536.1528} C_DIS
LIN {X 8.8897,Y -137.5915,Z 167,A -83.4245,B 10.6622,C 0.3069,E1 10.6813,E2 534.2189} C_DIS
LIN {X 14.7083,Y -137.0909,Z 167,A -81.7682,B 10.6617,C 0.3247,E1 10.6856,E2 532.6612} C_DIS
LIN {X 18.8772,Y -136.5807,Z 167,A -79.9886,B 10.6617,C 0.323,E1 10.6906,E2 530.8762} C_DIS
LIN {X 23.0957,Y -135.9301,Z 167,A -77.3892,B 10.6623,C 0.3016,E1 10.6981,E2 528.1685} C_DIS
LIN {X 29.4042,Y -134.706,Z 167,A -75.5456,B 10.6618,C 0.3201,E1 10.7028,E2 526.4305} C_DIS
LIN {X 33.272,Y -133.8044,Z 167,A -73.9,B 10.6618,C 0.3189,E1 10.7072,E2 524.7844} C_DIS
LIN {X 36.8635,Y -132.8584,Z 167,A -72.5419,B 10.6618,C 0.3221,E1 10.7108,E2 523.449} C_DIS
LIN {X 40.1037,Y -131.9164,Z 167,A -71.0357,B 10.6618,C 0.3181,E1 10.7149,E2 521.9283} C_DIS
LIN {X 43.3549,Y -130.8838,Z 167,A -69.6089,B 10.6619,C 0.3165,E1 10.7187,E2 520.4993} C_DIS
LIN {X 46.5267,Y -129.7902,Z 167,A -68.2333,B 10.6619,C 0.3154,E1 10.7223,E2 519.1249} C_DIS
LIN {X 49.8389,Y -128.5545,Z 167,A -66.6858,B 10.662,C 0.3117,E1 10.7264,E2 517.5662} C_DIS
LIN {X 53.5671,Y -127.047,Z 167,A -65.0755,B 10.662,C 0.3112,E1 10.7305,E2 515.9623} C_DIS
LIN {X 57.3256,Y -125.3965,Z 167,A -63.4969,B 10.662,C 0.3121,E1 10.7345,E2 514.3987} C_DIS
LIN {X 62.8252,Y -122.7323,Z 167,A -61.2868,B 10.6619,C 0.3169,E1 10.74,E2 512.2288} C_DIS
LIN {X 67.5718,Y -120.1863,Z 167,A -58.6472,B 10.6623,C 0.3035,E1 10.7466,E2 509.5359} C_DIS
LIN {X 71.4967,Y -117.8934,Z 167,A -56.2734,B 10.6627,C 0.288,E1 10.7524,E2 507.0975} C_DIS
LIN {X 75.3373,Y -115.4776,Z 167,A -54.8191,B 10.6625,C 0.2959,E1 10.7557,E2 505.6974} C_DIS
LIN {X 78.9594,Y -113.0317,Z 167,A -53.2401,B 10.6625,C 0.2988,E1 10.7593,E2 504.1471} C_DIS
LIN {X 82.8185,Y -110.2355,Z 167,A -51.0821,B 10.6626,C 0.2906,E1 10.7642,E2 501.9643} C_DIS
LIN {X 86.0809,Y -107.7072,Z 167,A -49.5349,B 10.6626,C 0.2916,E1 10.7676,E2 500.437} C_DIS
LIN {X 88.8056,Y -105.4719,Z 167,A -47.9157,B 10.6628,C 0.2848,E1 10.7711,E2 498.7964} C_DIS
LIN {X 93.7181,Y -101.1321,Z 167,A -45.1897,B 10.6629,C 0.2791,E1 10.7768,E2 496.0674} C_DIS
LIN {X 96.7379,Y -98.2473,Z 167,A -43.4614,B 10.663,C 0.2756,E1 10.7802,E2 494.3381} C_DIS
LIN {X 99.9754,Y -94.9515,Z 167,A -41.8315,B 10.663,C 0.279,E1 10.7833,E2 492.7436} C_DIS
LIN {X 102.6288,Y -92.0762,Z 167,A -39.779,B 10.6633,C 0.2642,E1 10.7873,E2 490.6343} C_DIS
LIN {X 104.8395,Y -89.5514,Z 167,A -38.3186,B 10.6634,C 0.2592,E1 10.7899,E2 489.1639} C_DIS
LIN {X 107.2359,Y -86.667,Z 167,A -37.0629,B 10.6634,C 0.2635,E1 10.7921,E2 487.9455} C_DIS
LIN {X 109.6928,Y -83.536,Z 167,A -34.9137,B 10.6637,C 0.2465,E1 10.7958,E2 485.7305} C_DIS
LIN {X 112.6583,Y -79.4908,Z 167,A -33.3403,B 10.6635,C 0.2549,E1 10.7983,E2 484.2209} C_DIS
LIN {X 115.2286,Y -75.717,Z 167,A -31.5358,B 10.6635,C 0.2526,E1 10.8011,E2 482.4263} C_DIS
LIN {X 117.5304,Y -72.0923,Z 167,A -29.5439,B 10.6638,C 0.2425,E1 10.804,E2 480.4057} C_DIS
LIN {X 119.1957,Y -69.3047,Z 167,A -28.3781,B 10.6638,C 0.2439,E1 10.8057,E2 479.262} C_DIS
LIN {X 121.3935,Y -65.3783,Z 167,A -26.5473,B 10.6638,C 0.24,E1 10.8081,E2 477.4342} C_DIS
LIN {X 124.2764,Y -59.7127,Z 167,A -24.0991,B 10.6639,C 0.2381,E1 10.8112,E2 475.0077} C_DIS
LIN {X 126.5041,Y -54.8351,Z 167,A -21.8553,B 10.6641,C 0.2317,E1 10.8137,E2 472.7595} C_DIS
LIN {X 127.6658,Y -52.0761,Z 167,A -20.5203,B 10.6641,C 0.2258,E1 10.8152,E2 471.4115} C_DIS
LIN {X 129.3462,Y -47.751,Z 167,A -18.6107,B 10.6643,C 0.221,E1 10.817,E2 469.5021} C_DIS
LIN {X 130.6993,Y -43.9089,Z 167,A -16.9665,B 10.6643,C 0.2175,E1 10.8185,E2 467.8623} C_DIS
LIN {X 131.7376,Y -40.688,Z 167,A -15.6134,B 10.6644,C 0.2149,E1 10.8197,E2 466.5143} C_DIS
LIN {X 132.7435,Y -37.2743,Z 167,A -14.2445,B 10.6644,C 0.2136,E1 10.8207,E2 465.1579} C_DIS
LIN {X 133.8483,Y -33.0984,Z 167,A -12.354,B 10.6646,C 0.206,E1 10.822,E2 463.2533} C_DIS
LIN {X 134.7001,Y -29.4316,Z 167,A -10.8376,B 10.6646,C 0.2027,E1 10.823,E2 461.7413} C_DIS
LIN {X 135.7608,Y -24.0684,Z 167,A -8.5445,B 10.6648,C 0.1956,E1 10.8242,E2 459.443} C_DIS
LIN {X 136.9307,Y -16.1328,Z 167,A -5.3992,B 10.6648,C 0.1909,E1 10.8254,E2 456.3183} C_DIS
LIN {X 137.5452,Y -9.5814,Z 167,A -2.1097,B 10.6652,C 0.168,E1 10.8261,E2 452.9549} C_DIS
LIN {X 137.7903,Y -4.9323,Z 167,A -0.6725,B 10.6652,C 0.1757,E1 10.8263,E2 451.5795} C_DIS
LIN {X 137.8741,Y -1.0901,Z 167,A 1.5195,B 10.6654,C 0.155,E1 10.8263,E2 449.3095} C_DIS
LIN {X 137.8088,Y 4.3979,Z 167,A 3.0192,B 10.6652,C 0.1693,E1 10.8263,E2 447.9077} C_DIS
LIN {X 137.3397,Y 12.1821,Z 167,A 6.2326,B 10.6654,C 0.1606,E1 10.8257,E2 444.6948} C_DIS
LIN {X 136.7303,Y 17.7511,Z 167,A 8.602,B 10.6654,C 0.1527,E1 10.8249,E2 442.3179} C_DIS
LIN {X 136.1367,Y 21.8545,Z 167,A 10.3811,B 10.6656,C 0.1463,E1 10.8241,E2 440.5301} C_DIS
LIN {X 135.4427,Y 25.7974,Z 167,A 11.7084,B 10.6656,C 0.1504,E1 10.8235,E2 439.2439} C_DIS
LIN {X 134.5979,Y 29.9047,Z 167,A 13.7354,B 10.6656,C 0.1379,E1 10.8223,E2 437.1794} C_DIS
LIN {X 133.8116,Y 33.2438,Z 167,A 15.1522,B 10.6657,C 0.1341,E1 10.8214,E2 435.7624} C_DIS
LIN {X 132.8301,Y 36.9648,Z 167,A 16.5899,B 10.6657,C 0.1339,E1 10.8203,E2 434.3438} C_DIS
LIN {X 131.8472,Y 40.3297,Z 167,A 18.1071,B 10.6657,C 0.1282,E1 10.8191,E2 432.8176} C_DIS
LIN {X 130.5429,Y 44.3779,Z 167,A 19.9323,B 10.6659,C 0.1218,E1 10.8175,E2 430.9839} C_DIS
LIN {X 128.4343,Y 50.148,Z 167,A 22.3882,B 10.6659,C 0.1174,E1 10.8151,E2 428.5381} C_DIS
LIN {X 126.7863,Y 54.1824,Z 167,A 24.0631,B 10.6659,C 0.1162,E1 10.8133,E2 426.8792} C_DIS
LIN {X 125.2879,Y 57.5603,Z 167,A 25.6439,B 10.6659,C 0.1109,E1 10.8115,E2 425.2914} C_DIS
LIN {X 123.4721,Y 61.3591,Z 167,A 27.4536,B 10.666,C 0.1048,E1 10.8093,E2 423.4729} C_DIS
LIN {X 121.3895,Y 65.3858,Z 167,A 29.0769,B 10.666,C 0.1068,E1 10.8072,E2 421.8813} C_DIS
LIN {X 118.5264,Y 70.443,Z 167,A 31.6725,B 10.6661,C 0.096,E1 10.8036,E2 419.2615} C_DIS
LIN {X 116.2801,Y 74.0926,Z 167,A 33.482,B 10.6661,C 0.0909,E1 10.8009,E2 417.4473} C_DIS
LIN {X 114.0258,Y 77.517,Z 167,A 35.1423,B 10.6661,C 0.0879,E1 10.7983,E2 415.7915} C_DIS
LIN {X 111.5325,Y 81.0631,Z 167,A 36.8887,B 10.6662,C 0.0851,E1 10.7955,E2 414.0509} C_DIS
LIN {X 109.8127,Y 83.3788,Z 167,A 38.39,B 10.6662,C 0.0746,E1 10.7929,E2 412.5109} C_DIS
LIN {X 107.5183,Y 86.3168,Z 167,A 39.4533,B 10.6662,C 0.0836,E1 10.7911,E2 411.508} C_DIS
LIN {X 105.2613,Y 89.0553,Z 167,A 41.1394,B 10.6662,C 0.0749,E1 10.7881,E2 409.7946} C_DIS
LIN {X 103.1837,Y 91.454,Z 167,A 43.3365,B 10.6664,C 0.0494,E1 10.7838,E2 407.4855} C_DIS
LIN {X 98.1856,Y 96.8009,Z 167,A 45.4004,B 10.6664,C 0.0683,E1 10.78,E2 405.5446} C_DIS
LIN {X 94.3568,Y 100.5366,Z 167,A 47.6445,B 10.6664,C 0.0633,E1 10.7755,E2 403.297} C_DIS
LIN {X 90.9712,Y 103.6103,Z 167,A 49.3958,B 10.6664,C 0.0635,E1 10.7718,E2 401.5637} C_DIS
LIN {X 87.3983,Y 106.6408,Z 167,A 51.4338,B 10.6664,C 0.0576,E1 10.7675,E2 399.5138} C_DIS
LIN {X 83.7485,Y 109.5302,Z 167,A 53.274,B 10.6664,C 0.0566,E1 10.7634,E2 397.6849} C_DIS
LIN {X 80.4681,Y 111.9629,Z 167,A 55.0749,B 10.6664,C 0.0511,E1 10.7593,E2 395.8706} C_DIS
LIN {X 76.7148,Y 114.5669,Z 167,A 56.9414,B 10.6664,C 0.0488,E1 10.755,E2 394.0078} C_DIS
LIN {X 72.9508,Y 116.9995,Z 167,A 58.7823,B 10.6664,C 0.0465,E1 10.7507,E2 392.1693} C_DIS
LIN {X 68.8897,Y 119.436,Z 167,A 60.6793,B 10.6664,C 0.0454,E1 10.7461,E2 390.2809} C_DIS
LIN {X 65.2245,Y 121.4762,Z 167,A 62.5077,B 10.6664,C 0.041,E1 10.7416,E2 388.4417} C_DIS
LIN {X 61.3363,Y 123.4833,Z 167,A 64.0481,B 10.6664,C 0.0454,E1 10.7379,E2 386.9358} C_DIS
LIN {X 58.2788,Y 124.9557,Z 167,A 65.6131,B 10.6664,C 0.04,E1 10.7339,E2 385.3515} C_DIS
LIN {X 55.3828,Y 126.2673,Z 167,A 66.8526,B 10.6664,C 0.0404,E1 10.7308,E2 384.1222} C_DIS
LIN {X 51.4358,Y 127.9239,Z 167,A 68.625,B 10.6664,C 0.0387,E1 10.7262,E2 382.3507} C_DIS
LIN {X 48.5274,Y 129.0554,Z 167,A 69.9815,B 10.6664,C 0.0359,E1 10.7226,E2 380.9869} C_DIS
LIN {X 44.9688,Y 130.3381,Z 167,A 71.5026,B 10.6664,C 0.0357,E1 10.7186,E2 379.4722} C_DIS
LIN {X 41.2282,Y 131.5713,Z 167,A 73.1774,B 10.6665,C 0.0334,E1 10.7142,E2 377.793} C_DIS
LIN {X 37.4712,Y 132.6884,Z 167,A 74.6126,B 10.6665,C 0.0367,E1 10.7104,E2 376.3821} C_DIS
LIN {X 32.074,Y 134.0952,Z 167,A 77.1142,B 10.6665,C 0.0308,E1 10.7036,E2 373.8582} C_DIS
LIN {X 28.0682,Y 134.9916,Z 167,A 78.8151,B 10.6665,C 0.03,E1 10.6989,E2 372.1584} C_DIS
LIN {X 22.7522,Y 135.9874,Z 167,A 81.6417,B 10.6665,C 0.0152,E1 10.6909,E2 369.26} C_DIS
LIN {X 17.7062,Y 136.7362,Z 167,A 83.1975,B 10.6665,C 0.0278,E1 10.6868,E2 367.7754} C_DIS
LIN {X 14.3662,Y 137.1277,Z 167,A 85.1353,B 10.6665,C 0.0147,E1 10.6813,E2 365.7706} C_DIS
LIN {X 9.3254,Y 137.5638,Z 167,A 86.5521,B 10.6665,C 0.0304,E1 10.6776,E2 364.4403} C_DIS
LIN {X 3.8282,Y 137.8247,Z 167,A 88.9481,B 10.6665,C 0.0277,E1 10.6708,E2 362.0317} C_DIS
LIN {X -4.3301,Y 137.8107,Z 167,A 92.0955,B 10.6665,C 0.0335,E1 10.6622,E2 358.9162} C_DIS
LIN {X -8.2676,Y 137.6298,Z 167,A 94.087,B 10.6665,C 0.0258,E1 10.6565,E2 356.8817} C_DIS
LIN {X -11.9271,Y 137.3613,Z 167,A 96.0896,B 10.6665,C 0.0153,E1 10.6507,E2 354.8204} C_DIS
LIN {X -16.9844,Y 136.8291,Z 167,A 97.7918,B 10.6665,C 0.0255,E1 10.6462,E2 353.1709} C_DIS
LIN {X -21.2431,Y 136.2314,Z 167,A 99.3823,B 10.6665,C 0.0308,E1 10.6418,E2 351.6058} C_DIS
LIN {X -25.2277,Y 135.5516,Z 167,A 101.1919,B 10.6665,C 0.0288,E1 10.6368,E2 349.7812} C_DIS
LIN {X -30.0282,Y 134.5697,Z 167,A 103.2366,B 10.6665,C 0.03,E1 10.6312,E2 347.7368} C_DIS
LIN {X -33.7043,Y 133.6947,Z 167,A 104.6597,B 10.6665,C 0.0344,E1 10.6274,E2 346.3329} C_DIS
LIN {X -36.9991,Y 132.8205,Z 167,A 106.0933,B 10.6665,C 0.0352,E1 10.6236,E2 344.8983} C_DIS
LIN {X -39.726,Y 132.032,Z 167,A 107.3303,B 10.6665,C 0.035,E1 10.6202,E2 343.655} C_DIS
LIN {X -44.2364,Y 130.5903,Z 167,A 109.6348,B 10.6665,C 0.0294,E1 10.614,E2 341.3102} C_DIS
LIN {X -47.693,Y 129.3679,Z 167,A 110.9105,B 10.6665,C 0.0365,E1 10.6108,E2 340.0665} C_DIS
LIN {X -51.8158,Y 127.7708,Z 167,A 112.711,B 10.6665,C 0.0394,E1 10.6061,E2 338.272} C_DIS
LIN {X -55.815,Y 126.0758,Z 167,A 114.5685,B 10.6665,C 0.0404,E1 10.6013,E2 336.4095} C_DIS
LIN {X -59.179,Y 124.5314,Z 167,A 115.9665,B 10.6665,C 0.0454,E1 10.5978,E2 335.0302} C_DIS
LIN {X -64.2671,Y 121.9832,Z 167,A 118.4154,B 10.6665,C 0.0468,E1 10.5917,E2 332.5729} C_DIS
LIN {X -67.9327,Y 119.9834,Z 167,A 120.2623,B 10.6665,C 0.047,E1 10.5872,E2 330.7139} C_DIS
LIN {X -71.8646,Y 117.67,Z 167,A 122.4203,B 10.6665,C 0.0443,E1 10.582,E2 328.525} C_DIS
LIN {X -74.9753,Y 115.7126,Z 167,A 124.6493,B 10.6665,C 0.0317,E1 10.5766,E2 326.2094} C_DIS
LIN {X -81.0744,Y 111.5243,Z 167,A 126.5548,B 10.6664,C 0.0621,E1 10.5726,E2 324.453} C_DIS
LIN {X -86.2296,Y 107.5883,Z 167,A 130.0804,B 10.6664,C 0.0495,E1 10.5646,E2 320.8268} C_DIS
LIN {X -90.315,Y 104.1829,Z 167,A 131.7596,B 10.6664,C 0.065,E1 10.5612,E2 319.2162} C_DIS
LIN {X -96.1433,Y 98.8294,Z 167,A 135.8857,B 10.6664,C 0.0542,E1 10.5526,E2 314.9887} C_DIS
LIN {X -100.7916,Y 94.0838,Z 167,A 137.8128,B 10.6663,C 0.0776,E1 10.5491,E2 313.1689} C_DIS
LIN {X -104.8286,Y 89.5638,Z 167,A 140.3427,B 10.6663,C 0.083,E1 10.5444,E2 310.6403} C_DIS
LIN {X -107.3876,Y 86.4789,Z 167,A 142.0216,B 10.6663,C 0.0866,E1 10.5415,E2 308.9615} C_DIS
LIN {X -109.8891,Y 83.2776,Z 167,A 143.5992,B 10.6662,C 0.0928,E1 10.5388,E2 307.3995} C_DIS
LIN {X -112.3379,Y 79.9436,Z 167,A 145.5393,B 10.6662,C 0.0924,E1 10.5356,E2 305.4338} C_DIS
LIN {X -114.8063,Y 76.3561,Z 167,A 147.3573,B 10.6662,C 0.0967,E1 10.5327,E2 303.6168} C_DIS
LIN {X -117.2422,Y 72.5608,Z 167,A 149.2576,B 10.6661,C 0.1009,E1 10.5299,E2 301.7153} C_DIS
LIN {X -119.4993,Y 68.7803,Z 167,A 151.0926,B 10.6661,C 0.1055,E1 10.5273,E2 299.8816} C_DIS
LIN {X -121.589,Y 65.0145,Z 167,A 152.8458,B 10.666,C 0.1109,E1 10.525,E2 298.135} C_DIS
LIN {X -124.752,Y 58.7171,Z 167,A 155.7936,B 10.666,C 0.1183,E1 10.5214,E2 295.1881} C_DIS
LIN {X -126.2887,Y 55.3333,Z 167,A 157.4352,B 10.6659,C 0.1205,E1 10.5195,E2 293.5362} C_DIS
LIN {X -127.5474,Y 52.3689,Z 167,A 158.6971,B 10.6659,C 0.1257,E1 10.5181,E2 292.2852} C_DIS
LIN {X -129.4972,Y 47.3393,Z 167,A 160.8913,B 10.6657,C 0.1328,E1 10.516,E2 290.0995} C_DIS
LIN {X -130.3463,Y 44.9451,Z 167,A 162.4684,B 10.6658,C 0.1252,E1 10.5145,E2 288.4585} C_DIS
LIN {X -131.6165,Y 41.0838,Z 167,A 163.8796,B 10.6658,C 0.1356,E1 10.5133,E2 287.084} C_DIS
LIN {X -132.6906,Y 37.4633,Z 167,A 165.394,B 10.6656,C 0.1412,E1 10.5121,E2 285.5781} C_DIS
LIN {X -133.6014,Y 34.0717,Z 167,A 166.7331,B 10.6656,C 0.1478,E1 10.5112,E2 284.2556} C_DIS
LIN {X -134.4412,Y 30.5908,Z 167,A 168.4099,B 10.6656,C 0.1482,E1 10.5101,E2 282.5569} C_DIS
LIN {X -135.2797,Y 26.6497,Z 167,A 170.1721,B 10.6655,C 0.1513,E1 10.5091,E2 280.7856} C_DIS
LIN {X -135.9713,Y 22.8488,Z 167,A 171.6812,B 10.6654,C 0.1579,E1 10.5084,E2 279.2903} C_DIS
LIN {X -136.4864,Y 19.5371,Z 167,A 173.1146,B 10.6654,C 0.1611,E1 10.5078,E2 277.8532} C_DIS
LIN {X -137.0208,Y 15.3597,Z 167,A 174.7671,B 10.6652,C 0.1682,E1 10.5073,E2 276.2148} C_DIS
LIN {X -137.4585,Y 10.7597,Z 167,A 177.0446,B 10.6652,C 0.1666,E1 10.5067,E2 273.8946} C_DIS
LIN {X -137.7401,Y 6.2031,Z 167,A 178.8621,B 10.6652,C 0.1738,E1 10.5065,E2 272.0891} C_DIS
LIN {X -137.8717,Y 1.4845,Z 167,A -178.9672,B 10.6652,C 0.1754,E1 10.5064,E2 269.8942} C_DIS
LIN {X -137.8667,Y -1.8142,Z 167,A -177.8656,B 10.665,C 0.1848,E1 10.5064,E2 268.8277} C_DIS
LIN {X -137.6833,Y -7.333,Z 167,A -175.4312,B 10.665,C 0.1887,E1 10.5067,E2 266.3781} C_DIS
LIN {X -137.4047,Y -11.4128,Z 167,A -173.8101,B 10.6648,C 0.1952,E1 10.507,E2 264.7685} C_DIS
LIN {X -137.0735,Y -14.8702,Z 167,A -172.3418,B 10.6648,C 0.1989,E1 10.5074,E2 263.2985} C_DIS
LIN {X -136.5456,Y -19.1232,Z 167,A -170.5317,B 10.6646,C 0.2035,E1 10.5081,E2 261.4864} C_DIS
LIN {X -136.0094,Y -22.6204,Z 167,A -169.2002,B 10.6645,C 0.2105,E1 10.5087,E2 260.1737} C_DIS
LIN {X -135.4583,Y -25.7159,Z 167,A -167.8441,B 10.6645,C 0.2132,E1 10.5094,E2 258.8125} C_DIS
LIN {X -134.7686,Y -29.1143,Z 167,A -166.3249,B 10.6644,C 0.2158,E1 10.5102,E2 257.2848} C_DIS
LIN {X -134.0356,Y -32.3213,Z 167,A -164.9385,B 10.6644,C 0.2192,E1 10.5111,E2 255.8971} C_DIS
LIN {X -133.3418,Y -35.0769,Z 167,A -163.6341,B 10.6644,C 0.2201,E1 10.512,E2 254.5783} C_DIS
LIN {X -131.9602,Y -39.9606,Z 167,A -161.3443,B 10.6643,C 0.2222,E1 10.5138,E2 252.2674} C_DIS
LIN {X -130.3222,Y -45.0146,Z 167,A -159.2568,B 10.6641,C 0.2308,E1 10.5157,E2 250.1969} C_DIS
LIN {X -128.8331,Y -49.1207,Z 167,A -157.4282,B 10.664,C 0.2354,E1 10.5175,E2 248.3682} C_DIS
LIN {X -127.4378,Y -52.6312,Z 167,A -155.8361,B 10.664,C 0.2392,E1 10.5191,E2 246.7744} C_DIS
LIN {X -125.9571,Y -56.0803,Z 167,A -154.3119,B 10.6638,C 0.244,E1 10.5208,E2 245.2558} C_DIS
LIN {X -124.5153,Y -59.2125,Z 167,A -152.9013,B 10.6637,C 0.2482,E1 10.5225,E2 243.8491} C_DIS
LIN {X -123.0219,Y -62.2564,Z 167,A -151.4564,B 10.6637,C 0.2511,E1 10.5243,E2 242.4006} C_DIS
LIN {X -121.2884,Y -65.5739,Z 167,A -149.8672,B 10.6636,C 0.2544,E1 10.5264,E2 240.8082} C_DIS
LIN {X -119.3161,Y -69.0967,Z 167,A -148.1177,B 10.6635,C 0.2571,E1 10.5288,E2 239.0508} C_DIS
LIN {X -117.117,Y -72.762,Z 167,A -146.2803,B 10.6635,C 0.2601,E1 10.5315,E2 237.2068} C_DIS
LIN {X -114.6787,Y -76.5472,Z 167,A -144.4321,B 10.6633,C 0.2651,E1 10.5343,E2 235.3625} C_DIS
LIN {X -112.3981,Y -79.8594,Z 167,A -142.8581,B 10.6631,C 0.271,E1 10.5368,E2 233.8018} C_DIS
LIN {X -110.1507,Y -82.9309,Z 167,A -141.0935,B 10.6631,C 0.2708,E1 10.5398,E2 232.0149} C_DIS
LIN {X -107.458,Y -86.3916,Z 167,A -139.2394,B 10.6631,C 0.2742,E1 10.543,E2 230.1576} C_DIS
LIN {X -105.4156,Y -88.8726,Z 167,A -137.4037,B 10.6633,C 0.2664,E1 10.5465,E2 228.2586} C_DIS
LIN {X -102.1864,Y -92.5669,Z 167,A -135.8413,B 10.6629,C 0.2809,E1 10.5492,E2 226.7581} C_DIS
LIN {X -98.998,Y -95.9692,Z 167,A -133.9507,B 10.6628,C 0.2859,E1 10.5529,E2 224.8743} C_DIS
LIN {X -95.8684,Y -99.0955,Z 167,A -132.0274,B 10.6628,C 0.2877,E1 10.5567,E2 222.9409} C_DIS
LIN {X -92.415,Y -102.3243,Z 167,A -130.303,B 10.6625,C 0.2966,E1 10.5602,E2 221.2477} C_DIS
LIN {X -89.9728,Y -104.4776,Z 167,A -128.7469,B 10.6625,C 0.2947,E1 10.5635,E2 219.6662} C_DIS
LIN {X -87.025,Y -106.9458,Z 167,A -127.0953,B 10.6625,C 0.2963,E1 10.5671,E2 218.0082} C_DIS
LIN {X -83.6457,Y -109.6089,Z 167,A -125.2892,B 10.6625,C 0.299,E1 10.5711,E2 216.2002} C_DIS
LIN {X -80.0754,Y -112.2437,Z 167,A -123.4149,B 10.6623,C 0.3013,E1 10.5753,E2 214.3225} C_DIS
LIN {X -76.2486,Y -114.8781,Z 167,A -121.4957,B 10.6623,C 0.3045,E1 10.5798,E2 212.4051} C_DIS
LIN {X -72.5859,Y -117.2266,Z 167,A -119.6387,B 10.6623,C 0.3061,E1 10.5842,E2 210.5421} C_DIS
LIN {X -68.7974,Y -119.4894,Z 167,A -117.7936,B 10.6621,C 0.3084,E1 10.5886,E2 208.6957} C_DIS
LIN {X -64.883,Y -121.6596,Z 167,A -115.9495,B 10.6621,C 0.3111,E1 10.5931,E2 206.8538} C_DIS
LIN {X -61.5202,Y -123.3926,Z 167,A -114.3837,B 10.6621,C 0.3132,E1 10.597,E2 205.2888} C_DIS
LIN {X -58.554,Y -124.8285,Z 167,A -113.1048,B 10.6619,C 0.3168,E1 10.6002,E2 204.0215} C_DIS
LIN {X -53.8705,Y -126.9203,Z 167,A -110.8721,B 10.6619,C 0.3168,E1 10.606,E2 201.7759} C_DIS
LIN {X -50.2961,Y -128.3768,Z 167,A -109.2908,B 10.6619,C 0.3188,E1 10.6101,E2 200.1973} C_DIS
LIN {X -47.0984,Y -129.5841,Z 167,A -107.8205,B 10.6619,C 0.319,E1 10.6139,E2 198.7204} C_DIS
LIN {X -43.6211,Y -130.7952,Z 167,A -106.3484,B 10.6618,C 0.3215,E1 10.6178,E2 197.2556} C_DIS
LIN {X -40.5538,Y -131.7787,Z 167,A -104.4155,B 10.6621,C 0.3089,E1 10.6232,E2 195.2459} C_DIS
LIN {X -35.8216,Y -133.1431,Z 167,A -102.9454,B 10.6617,C 0.3235,E1 10.6269,E2 193.8499} C_DIS
LIN {X -32.3716,Y -134.0235,Z 167,A -101.4864,B 10.6617,C 0.3249,E1 10.6309,E2 192.3931} C_DIS
LIN {X -29.2893,Y -134.7308,Z 167,A -99.8023,B 10.6619,C 0.3169,E1 10.6356,E2 190.6612} C_DIS
LIN {X -25.7567,Y -135.4505,Z 167,A -97.6944,B 10.6623,C 0.3032,E1 10.6416,E2 188.4737} C_DIS
LIN {X -18.8942,Y -136.5783,Z 167,A -95.8454,B 10.6615,C 0.3286,E1 10.6464,E2 186.7587} C_DIS
LIN {X -13.0725,Y -137.2566,Z 167,A -93.3217,B 10.6615,C 0.3271,E1 10.6534,E2 184.2228} C_DIS
LIN {X -9.3734,Y -137.5604,Z 167,A -91.6946,B 10.6617,C 0.3252,E1 10.658,E2 182.5843} C_DIS
LIN {X -5.5542,Y -137.766,Z 167,A -90.2034,B 10.6616,C 0.3275,E1 10.6621,E2 181.1049} C_DIS
LIN {X 0.4955,Y -137.8772,Z 167,A -87.5993,B 10.6616,C 0.3252,E1 10.6694,E2 178.4882} C_DIS
LIN {X 0.4955,Y -137.8772,Z 167,A -87.5993,B 10.6616,C 0.3252,E1 10.6694,E2 178.4882} C_DIS
Enddeposition()
LIN {X 0.9856,Y -138.7815,Z 167,A -87.567,B 10.3436,C 0.3473,E1 10.3518,E2 178.6059} C_DIS
Startdeposition()
$VEL.CP = VEL_PRINT
LIN {X -3.3354,Y -138.7543,Z 167,A -89.8083,B 10.3432,C 0.3581,E1 10.3454,E2 180.9072} C_DIS
LIN {X -6.9702,Y -138.6182,Z 167,A -91.3044,B 10.3432,C 0.358,E1 10.3412,E2 182.4033} C_DIS
LIN {X -11.276,Y -138.3351,Z 167,A -92.8637,B 10.3434,C 0.3528,E1 10.337,E2 183.9348} C_DIS
LIN {X -14.4705,Y -138.0373,Z 167,A -94.8058,B 10.3429,C 0.3666,E1 10.3314,E2 185.9563} C_DIS
LIN {X -18.684,Y -137.5314,Z 167,A -96.2217,B 10.3432,C 0.3586,E1 10.3276,E2 187.3301} C_DIS
LIN {X -22.8127,Y -136.9055,Z 167,A -97.9843,B 10.3432,C 0.3588,E1 10.3227,E2 189.0981} C_DIS
LIN {X -30.4007,Y -135.4237,Z 167,A -101.0939,B 10.3433,C 0.3555,E1 10.3142,E2 192.1981} C_DIS
LIN {X -34.2865,Y -134.4915,Z 167,A -103.1293,B 10.3431,C 0.3631,E1 10.3085,E2 194.283} C_DIS
LIN {X -38.3529,Y -133.3904,Z 167,A -104.4657,B 10.3434,C 0.3531,E1 10.3051,E2 195.5685} C_DIS
LIN {X -41.694,Y -132.3836,Z 167,A -106.0039,B 10.3434,C 0.3542,E1 10.3009,E2 197.1194} C_DIS
LIN {X -44.976,Y -131.3046,Z 167,A -107.1856,B 10.3436,C 0.3476,E1 10.2979,E2 198.2701} C_DIS
LIN {X -48.1993,Y -130.1559,Z 167,A -108.807,B 10.3435,C 0.351,E1 10.2936,E2 199.9183} C_DIS
LIN {X -51.3843,Y -128.9318,Z 167,A -110.1236,B 10.3435,C 0.3476,E1 10.2902,E2 201.2233} C_DIS
LIN {X -54.8432,Y -127.498,Z 167,A -111.7093,B 10.3436,C 0.3469,E1 10.2861,E2 202.8142} C_DIS
LIN {X -59.9793,Y -125.1637,Z 167,A -113.9735,B 10.3437,C 0.3429,E1 10.2804,E2 205.0701} C_DIS
LIN {X -62.5734,Y -123.8879,Z 167,A -115.2818,B 10.3437,C 0.344,E1 10.2771,E2 206.3931} C_DIS
LIN {X -66.1205,Y -122.0337,Z 167,A -117.0216,B 10.3437,C 0.3438,E1 10.2727,E2 208.144} C_DIS
LIN {X -69.9994,Y -119.8507,Z 167,A -118.8704,B 10.3437,C 0.3415,E1 10.2683,E2 209.994} C_DIS
LIN {X -73.8268,Y -117.5317,Z 167,A -120.6966,B 10.3439,C 0.3384,E1 10.2639,E2 211.8173} C_DIS
LIN {X -77.4756,Y -115.1594,Z 167,A -122.5458,B 10.3439,C 0.3368,E1 10.2596,E2 213.673} C_DIS
LIN {X -81.2569,Y -112.5228,Z 167,A -124.4392,B 10.344,C 0.3336,E1 10.2553,E2 215.5647} C_DIS
LIN {X -84.7731,Y -109.8982,Z 167,A -126.3004,B 10.3441,C 0.3316,E1 10.2511,E2 217.4319} C_DIS
LIN {X -88.4137,Y -106.9908,Z 167,A -128.1889,B 10.3442,C 0.3275,E1 10.2471,E2 219.3154} C_DIS
LIN {X -91.5954,Y -104.2801,Z 167,A -129.9613,B 10.3442,C 0.3253,E1 10.2433,E2 221.0932} C_DIS
LIN {X -95.0078,Y -101.1811,Z 167,A -131.8971,B 10.3444,C 0.3224,E1 10.2393,E2 223.0326} C_DIS
LIN {X -98.1012,Y -98.1846,Z 167,A -133.6805,B 10.3444,C 0.319,E1 10.2358,E2 224.816} C_DIS
LIN {X -101.2315,Y -94.9544,Z 167,A -135.8545,B 10.3444,C 0.3217,E1 10.2315,E2 227.0292} C_DIS
LIN {X -103.8476,Y -92.0848,Z 167,A -137.4592,B 10.3445,C 0.3183,E1 10.2285,E2 228.6335} C_DIS
LIN {X -106.3753,Y -89.1532,Z 167,A -138.7381,B 10.3448,C 0.3084,E1 10.2263,E2 229.8714} C_DIS
LIN {X -108.7162,Y -86.2834,Z 167,A -140.2636,B 10.3449,C 0.305,E1 10.2237,E2 231.3957} C_DIS
LIN {X -110.4375,Y -84.0693,Z 167,A -141.4377,B 10.3449,C 0.3027,E1 10.2217,E2 232.5714} C_DIS
LIN {X -112.9352,Y -80.6824,Z 167,A -143.2496,B 10.3451,C 0.3002,E1 10.2187,E2 234.3918} C_DIS
LIN {X -115.62,Y -76.7862,Z 167,A -145.1808,B 10.3451,C 0.2951,E1 10.2156,E2 236.3191} C_DIS
LIN {X -117.9241,Y -73.1978,Z 167,A -146.9598,B 10.3453,C 0.2913,E1 10.213,E2 238.0993} C_DIS
LIN {X -120.1969,Y -69.4028,Z 167,A -148.837,B 10.3453,C 0.2878,E1 10.2103,E2 239.9819} C_DIS
LIN {X -122.3986,Y -65.4421,Z 167,A -150.7622,B 10.3455,C 0.2842,E1 10.2077,E2 241.9127} C_DIS
LIN {X -124.3256,Y -61.6985,Z 167,A -152.3966,B 10.3457,C 0.2776,E1 10.2057,E2 243.5329} C_DIS
LIN {X -125.8772,Y -58.4674,Z 167,A -153.9985,B 10.3457,C 0.2762,E1 10.2038,E2 245.1491} C_DIS
LIN {X -127.5672,Y -54.6831,Z 167,A -155.6715,B 10.3458,C 0.2709,E1 10.2019,E2 246.816} C_DIS
LIN {X -129.0455,Y -51.1024,Z 167,A -157.5815,B 10.3458,C 0.2728,E1 10.1999,E2 248.7639} C_DIS
LIN {X -130.2532,Y -47.9396,Z 167,A -158.8218,B 10.346,C 0.2659,E1 10.1987,E2 249.9835} C_DIS
LIN {X -131.7011,Y -43.7985,Z 167,A -160.5159,B 10.3462,C 0.2587,E1 10.1972,E2 251.6613} C_DIS
LIN {X -132.7057,Y -40.6533,Z 167,A -162.1964,B 10.3461,C 0.2611,E1 10.1957,E2 253.3805} C_DIS
LIN {X -133.6372,Y -37.4782,Z 167,A -163.3061,B 10.3463,C 0.2523,E1 10.1949,E2 254.457} C_DIS
LIN {X -134.481,Y -34.328,Z 167,A -164.664,B 10.3464,C 0.2488,E1 10.194,E2 255.8152} C_DIS
LIN {X -135.2608,Y -31.114,Z 167,A -166.0194,B 10.3464,C 0.2447,E1 10.1931,E2 257.1682} C_DIS
LIN {X -135.989,Y -27.7582,Z 167,A -167.4557,B 10.3466,C 0.241,E1 10.1923,E2 258.6056} C_DIS
LIN {X -136.6479,Y -24.3087,Z 167,A -168.9592,B 10.3466,C 0.2379,E1 10.1915,E2 260.1146} C_DIS
LIN {X -137.2663,Y -20.5428,Z 167,A -170.6897,B 10.3466,C 0.2364,E1 10.1907,E2 261.8631} C_DIS
LIN {X -137.7991,Y -16.5825,Z 167,A -172.2125,B 10.3468,C 0.2292,E1 10.1902,E2 263.3685} C_DIS
LIN {X -138.1575,Y -13.2691,Z 167,A -173.6219,B 10.3469,C 0.2259,E1 10.1898,E2 264.7808} C_DIS
LIN {X -138.4789,Y -9.3658,Z 167,A -175.217,B 10.347,C 0.2208,E1 10.1895,E2 266.3717} C_DIS
LIN {X -138.6357,Y -6.6227,Z 167,A -176.6435,B 10.347,C 0.2231,E1 10.1893,E2 267.8334} C_DIS
LIN {X -138.7675,Y -2.7131,Z 167,A -178.6977,B 10.3469,C 0.2268,E1 10.1892,E2 269.9405} C_DIS
LIN {X -138.7711,Y 2.4961,Z 167,A 179.7668,B 10.3473,C 0.2087,E1 10.1892,E2 271.3976} C_DIS
LIN {X -138.6663,Y 5.9635,Z 167,A 178.0359,B 10.3473,C 0.2103,E1 10.1894,E2 273.1643} C_DIS
LIN {X -138.484,Y 9.2925,Z 167,A 176.9549,B 10.3474,C 0.2006,E1 10.1896,E2 274.2072} C_DIS
LIN {X -138.1448,Y 13.4018,Z 167,A 175.0598,B 10.3474,C 0.1993,E1 10.1901,E2 276.1245} C_DIS
LIN {X -137.6563,Y 17.7314,Z 167,A 173.3573,B 10.3476,C 0.1922,E1 10.1906,E2 277.8132} C_DIS
LIN {X -137.1742,Y 21.1375,Z 167,A 171.9185,B 10.3476,C 0.1885,E1 10.1912,E2 279.2527} C_DIS
LIN {X -136.5717,Y 24.7343,Z 167,A 170.3747,B 10.3477,C 0.1849,E1 10.192,E2 280.7998} C_DIS
LIN {X -135.7985,Y 28.6821,Z 167,A 168.6095,B 10.3477,C 0.1821,E1 10.1929,E2 282.5762} C_DIS
LIN {X -135.0306,Y 32.1006,Z 167,A 167.3974,B 10.3479,C 0.1734,E1 10.1937,E2 283.7576} C_DIS
LIN {X -134.2436,Y 35.2483,Z 167,A 165.82,B 10.3479,C 0.1742,E1 10.1948,E2 285.3631} C_DIS
LIN {X -133.2369,Y 38.8771,Z 167,A 164.313,B 10.3479,C 0.1689,E1 10.1959,E2 286.8625} C_DIS
LIN {X -131.9837,Y 42.9451,Z 167,A 162.0919,B 10.3479,C 0.1729,E1 10.1979,E2 289.1392} C_DIS
LIN {X -130.6863,Y 46.7407,Z 167,A 160.879,B 10.3481,C 0.1598,E1 10.199,E2 290.2955} C_DIS
LIN {X -128.4924,Y 52.4745,Z 167,A 158.2381,B 10.3482,C 0.1549,E1 10.2016,E2 292.9468} C_DIS
LIN {X -126.9775,Y 56.0414,Z 167,A 156.73,B 10.3483,C 0.1488,E1 10.2033,E2 294.4418} C_DIS
LIN {X -125.8412,Y 58.5453,Z 167,A 155.2782,B 10.3483,C 0.1519,E1 10.205,E2 295.9315} C_DIS
LIN {X -123.2349,Y 63.8527,Z 167,A 152.9561,B 10.3483,C 0.1431,E1 10.2079,E2 298.2363} C_DIS
LIN {X -121.1406,Y 67.7425,Z 167,A 151.0746,B 10.3484,C 0.1395,E1 10.2105,E2 300.1229} C_DIS
LIN {X -118.9666,Y 71.492,Z 167,A 149.2624,B 10.3484,C 0.1354,E1 10.213,E2 301.936} C_DIS
LIN {X -116.551,Y 75.3654,Z 167,A 147.369,B 10.3485,C 0.1309,E1 10.2159,E2 303.8285} C_DIS
LIN {X -114.0924,Y 79.038,Z 167,A 145.654,B 10.3486,C 0.1242,E1 10.2185,E2 305.528} C_DIS
LIN {X -111.8827,Y 82.1356,Z 167,A 143.8596,B 10.3486,C 0.1249,E1 10.2215,E2 307.3483} C_DIS
LIN {X -109.0187,Y 85.9009,Z 167,A 141.9534,B 10.3486,C 0.1194,E1 10.2248,E2 309.2467} C_DIS
LIN {X -105.7437,Y 89.9014,Z 167,A 139.32,B 10.3486,C 0.1244,E1 10.2296,E2 311.9391} C_DIS
LIN {X -102.5141,Y 93.5682,Z 167,A 137.7515,B 10.3488,C 0.111,E1 10.2324,E2 313.4505} C_DIS
LIN {X -99.3083,Y 96.9636,Z 167,A 135.4627,B 10.3488,C 0.1141,E1 10.237,E2 315.7816} C_DIS
LIN {X -96.3712,Y 99.8832,Z 167,A 133.7926,B 10.3488,C 0.1098,E1 10.2403,E2 317.4451} C_DIS
LIN {X -93.5518,Y 102.529,Z 167,A 132.4893,B 10.3488,C 0.1007,E1 10.2429,E2 318.7109} C_DIS
LIN {X -90.2041,Y 105.4864,Z 167,A 130.7096,B 10.3489,C 0.0958,E1 10.2466,E2 320.4809} C_DIS
LIN {X -86.326,Y 108.6822,Z 167,A 128.0939,B 10.3489,C 0.1028,E1 10.2524,E2 323.1609} C_DIS
LIN {X -82.7149,Y 111.4554,Z 167,A 126.6396,B 10.3489,C 0.0909,E1 10.2556,E2 324.5612} C_DIS
LIN {X -79.1745,Y 113.9974,Z 167,A 125.0479,B 10.349,C 0.0835,E1 10.2591,E2 326.1257} C_DIS
LIN {X -76.3326,Y 115.9195,Z 167,A 122.7382,B 10.3489,C 0.0994,E1 10.2648,E2 328.5435} C_DIS
LIN {X -71.4713,Y 118.9791,Z 167,A 120.963,B 10.349,C 0.0835,E1 10.2688,E2 330.2438} C_DIS
LIN {X -68.4869,Y 120.7214,Z 167,A 119.4177,B 10.349,C 0.0838,E1 10.2726,E2 331.8025} C_DIS
LIN {X -64.6603,Y 122.8109,Z 167,A 117.7376,B 10.349,C 0.0788,E1 10.2767,E2 333.4662} C_DIS
LIN {X -60.3265,Y 124.9978,Z 167,A 115.754,B 10.349,C 0.0757,E1 10.2817,E2 335.4457} C_DIS
LIN {X -57.1239,Y 126.4933,Z 167,A 114.4817,B 10.3491,C 0.07,E1 10.2848,E2 336.6937} C_DIS
LIN {X -54.6277,Y 127.5912,Z 167,A 113.0333,B 10.3491,C 0.0754,E1 10.2886,E2 338.1809} C_DIS
LIN {X -50.4527,Y 129.2982,Z 167,A 111.3514,B 10.3491,C 0.0695,E1 10.2929,E2 339.8391} C_DIS
LIN {X -47.4068,Y 130.4461,Z 167,A 109.9708,B 10.3491,C 0.0689,E1 10.2966,E2 341.2232} C_DIS
LIN {X -41.1216,Y 132.5624,Z 167,A 107.2151,B 10.3491,C 0.0666,E1 10.3039,E2 343.9792} C_DIS
LIN {X -37.7049,Y 133.5738,Z 167,A 105.8133,B 10.3491,C 0.0639,E1 10.3076,E2 345.3713} C_DIS
LIN {X -34.4641,Y 134.4464,Z 167,A 104.346,B 10.3491,C 0.0646,E1 10.3116,E2 346.8477} C_DIS
LIN {X -31.3032,Y 135.2176,Z 167,A 103.132,B 10.3491,C 0.0608,E1 10.3148,E2 348.0449} C_DIS
LIN {X -28.058,Y 135.928,Z 167,A 101.6212,B 10.3491,C 0.0629,E1 10.319,E2 349.572} C_DIS
LIN {X -24.5488,Y 136.6049,Z 167,A 100.2248,B 10.3491,C 0.0604,E1 10.3228,E2 350.9577} C_DIS
LIN {X -21.607,Y 137.1015,Z 167,A 98.5454,B 10.3491,C 0.0695,E1 10.3276,E2 352.6914} C_DIS
LIN {X -17.8034,Y 137.6468,Z 167,A 97.3971,B 10.3491,C 0.0593,E1 10.3306,E2 353.7851} C_DIS
LIN {X -11.569,Y 138.3103,Z 167,A 94.737,B 10.3491,C 0.06,E1 10.3381,E2 356.4526} C_DIS
LIN {X -7.8844,Y 138.5707,Z 167,A 93.0412,B 10.3491,C 0.0634,E1 10.3428,E2 358.1687} C_DIS
LIN {X -2.7247,Y 138.7672,Z 167,A 90.6687,B 10.3491,C 0.0685,E1 10.3495,E2 360.5697} C_DIS
LIN {X 1.3894,Y 138.7879,Z 167,A 89.3111,B 10.3491,C 0.0609,E1 10.3532,E2 361.8848} C_DIS
LIN {X 5.6656,Y 138.6779,Z 167,A 87.621,B 10.3491,C 0.0593,E1 10.3579,E2 363.5647} C_DIS
LIN {X 10.6977,Y 138.3814,Z 167,A 84.9426,B 10.3491,C 0.073,E1 10.3656,E2 366.3156} C_DIS
LIN {X 15.7637,Y 137.8968,Z 167,A 83.385,B 10.3491,C 0.0614,E1 10.3697,E2 367.8059} C_DIS
LIN {X 22.5393,Y 136.9511,Z 167,A 80.1733,B 10.3491,C 0.0713,E1 10.3787,E2 371.0644} C_DIS
LIN {X 26.8401,Y 136.1755,Z 167,A 78.7018,B 10.3491,C 0.0646,E1 10.3826,E2 372.4946} C_DIS
LIN {X 31.0193,Y 135.2824,Z 167,A 76.661,B 10.3491,C 0.072,E1 10.3883,E2 374.5689} C_DIS
LIN {X 34.9108,Y 134.3309,Z 167,A 75.1968,B 10.3491,C 0.0688,E1 10.3922,E2 376.0095} C_DIS
LIN {X 40.1011,Y 132.8747,Z 167,A 73.1541,B 10.3491,C 0.0663,E1 10.3976,E2 378.0293} C_DIS
LIN {X 43.8589,Y 131.681,Z 167,A 71.6456,B 10.3491,C 0.0649,E1 10.4015,E2 379.5228} C_DIS
LIN {X 46.9646,Y 130.6056,Z 167,A 70.2595,B 10.3491,C 0.0669,E1 10.4052,E2 380.9124} C_DIS
LIN {X 50.0852,Y 129.4411,Z 167,A 69.1015,B 10.3491,C 0.0632,E1 10.4082,E2 382.0433} C_DIS
LIN {X 52.9778,Y 128.2853,Z 167,A 67.6408,B 10.3491,C 0.0686,E1 10.412,E2 383.5258} C_DIS
LIN {X 56.3208,Y 126.8526,Z 167,A 66.0682,B 10.3491,C 0.072,E1 10.416,E2 385.1071} C_DIS
LIN {X 59.542,Y 125.3726,Z 167,A 64.5959,B 10.3491,C 0.074,E1 10.4198,E2 386.5805} C_DIS
LIN {X 62.7527,Y 123.7966,Z 167,A 63.1742,B 10.3491,C 0.0745,E1 10.4233,E2 387.9955} C_DIS
LIN {X 66.2107,Y 121.9845,Z 167,A 61.4595,B 10.3491,C 0.0792,E1 10.4276,E2 389.7231} C_DIS
LIN {X 70.2471,Y 119.7053,Z 167,A 59.5956,B 10.3491,C 0.0807,E1 10.4321,E2 391.581} C_DIS
LIN {X 73.9604,Y 117.4473,Z 167,A 57.8003,B 10.3491,C 0.0834,E1 10.4363,E2 393.3768} C_DIS
LIN {X 77.8045,Y 114.9368,Z 167,A 55.9203,B 10.3491,C 0.086,E1 10.4407,E2 395.2551} C_DIS
LIN {X 81.5951,Y 112.2776,Z 167,A 54.0357,B 10.349,C 0.0885,E1 10.445,E2 397.1368} C_DIS
LIN {X 85.2769,Y 109.5077,Z 167,A 52.0842,B 10.349,C 0.0931,E1 10.4493,E2 399.0949} C_DIS
LIN {X 87.7003,Y 107.5764,Z 167,A 50.5514,B 10.3489,C 0.1015,E1 10.4527,E2 400.6595} C_DIS
LIN {X 90.7708,Y 104.9987,Z 167,A 49.2719,B 10.3489,C 0.0955,E1 10.4553,E2 401.8929} C_DIS
LIN {X 93.8672,Y 102.2397,Z 167,A 47.7093,B 10.3489,C 0.0951,E1 10.4585,E2 403.4374} C_DIS
LIN {X 97.4902,Y 98.7919,Z 167,A 45.4579,B 10.3489,C 0.1038,E1 10.4631,E2 405.7129} C_DIS
LIN {X 104.0545,Y 91.8513,Z 167,A 41.5879,B 10.3488,C 0.1103,E1 10.4705,E2 409.5753} C_DIS
LIN {X 106.3706,Y 89.1589,Z 167,A 40.0884,B 10.3488,C 0.1144,E1 10.4732,E2 411.0797} C_DIS
LIN {X 110.7566,Y 83.6479,Z 167,A 37.28,B 10.3487,C 0.1185,E1 10.478,E2 413.8771} C_DIS
LIN {X 113.3669,Y 80.0747,Z 167,A 35.4462,B 10.3487,C 0.123,E1 10.481,E2 415.7129} C_DIS
LIN {X 116.0812,Y 76.087,Z 167,A 33.5294,B 10.3487,C 0.1259,E1 10.4839,E2 417.6214} C_DIS
LIN {X 118.0154,Y 73.0512,Z 167,A 31.7411,B 10.3485,C 0.1371,E1 10.4866,E2 419.4484} C_DIS
LIN {X 119.9571,Y 69.8168,Z 167,A 30.2315,B 10.3485,C 0.1398,E1 10.4887,E2 420.9531} C_DIS
LIN {X 121.7309,Y 66.6757,Z 167,A 28.9874,B 10.3485,C 0.1374,E1 10.4904,E2 422.1675} C_DIS
LIN {X 123.5594,Y 63.2186,Z 167,A 27.5254,B 10.3485,C 0.1377,E1 10.4922,E2 423.6114} C_DIS
LIN {X 124.9358,Y 60.4564,Z 167,A 26.0738,B 10.3483,C 0.1455,E1 10.4941,E2 425.0862} C_DIS
LIN {X 126.6415,Y 56.7925,Z 167,A 24.6329,B 10.3483,C 0.1441,E1 10.4957,E2 426.4997} C_DIS
LIN {X 128.4994,Y 52.457,Z 167,A 22.773,B 10.3483,C 0.1471,E1 10.4977,E2 428.3501} C_DIS
LIN {X 130.4662,Y 47.3512,Z 167,A 20.548,B 10.3483,C 0.1524,E1 10.4999,E2 430.5726} C_DIS
LIN {X 131.5811,Y 44.1588,Z 167,A 19.1476,B 10.3482,C 0.1563,E1 10.5012,E2 431.9747} C_DIS
LIN {X 132.5949,Y 41.0153,Z 167,A 17.8517,B 10.3482,C 0.1583,E1 10.5023,E2 433.2632} C_DIS
LIN {X 133.5981,Y 37.6178,Z 167,A 16.301,B 10.3481,C 0.1647,E1 10.5035,E2 434.8263} C_DIS
LIN {X 134.481,Y 34.328,Z 167,A 14.9467,B 10.3481,C 0.1673,E1 10.5045,E2 436.1751} C_DIS
LIN {X 135.4144,Y 30.4415,Z 167,A 13.1865,B 10.3479,C 0.1748,E1 10.5056,E2 437.9507} C_DIS
LIN {X 136.4467,Y 25.4213,Z 167,A 11.2009,B 10.3479,C 0.1775,E1 10.5067,E2 439.9218} C_DIS
LIN {X 137.1147,Y 21.5216,Z 167,A 9.4942,B 10.3477,C 0.1841,E1 10.5074,E2 441.6392} C_DIS
LIN {X 137.5645,Y 18.4316,Z 167,A 7.6864,B 10.3474,C 0.2012,E1 10.5081,E2 443.5136} C_DIS
LIN {X 138.1514,Y 13.3335,Z 167,A 6.1991,B 10.3476,C 0.1911,E1 10.5085,E2 444.9234} C_DIS
LIN {X 138.4161,Y 10.2269,Z 167,A 4.4884,B 10.3473,C 0.2058,E1 10.5089,E2 446.6888} C_DIS
LIN {X 138.6687,Y 5.9019,Z 167,A 3.0731,B 10.3474,C 0.2014,E1 10.5091,E2 448.0589} C_DIS
LIN {X 138.7933,Y -0.4332,Z 167,A 0.6027,B 10.3474,C 0.2053,E1 10.5091,E2 450.5134} C_DIS
LIN {X 138.739,Y -3.8841,Z 167,A -0.8071,B 10.3473,C 0.2091,E1 10.5091,E2 451.9228} C_DIS
LIN {X 138.5843,Y -7.6442,Z 167,A -2.5591,B 10.3471,C 0.2188,E1 10.5088,E2 453.7016} C_DIS
LIN {X 137.9863,Y -14.945,Z 167,A -5.3159,B 10.3471,C 0.2207,E1 10.5081,E2 456.4275} C_DIS
LIN {X 137.5,Y -18.916,Z 167,A -7.0436,B 10.3469,C 0.2275,E1 10.5075,E2 458.1667} C_DIS
LIN {X 136.8853,Y -22.9341,Z 167,A -9.2795,B 10.3464,C 0.2467,E1 10.5065,E2 460.4749} C_DIS
LIN {X 135.8418,Y -28.4814,Z 167,A -11.0267,B 10.3466,C 0.2385,E1 10.5055,E2 462.1511} C_DIS
LIN {X 135.1071,Y -31.783,Z 167,A -12.4736,B 10.3466,C 0.2438,E1 10.5046,E2 463.6059} C_DIS
LIN {X 133.8111,Y -36.8565,Z 167,A -14.4539,B 10.3465,C 0.2453,E1 10.5032,E2 465.5654} C_DIS
LIN {X 132.7855,Y -40.3924,Z 167,A -15.8659,B 10.3465,C 0.2468,E1 10.5021,E2 466.9653} C_DIS
LIN {X 131.6355,Y -43.9954,Z 167,A -17.41,B 10.3464,C 0.2507,E1 10.5008,E2 468.509} C_DIS
LIN {X 130.2948,Y -47.8266,Z 167,A -19.3993,B 10.346,C 0.2635,E1 10.4988,E2 470.5401} C_DIS
LIN {X 129.0695,Y -51.041,Z 167,A -20.5342,B 10.3461,C 0.2601,E1 10.4977,E2 471.6403} C_DIS
LIN {X 127.5092,Y -54.8173,Z 167,A -22.1711,B 10.3461,C 0.2634,E1 10.496,E2 473.2726} C_DIS
LIN {X 126.0796,Y -58.0297,Z 167,A -23.5749,B 10.346,C 0.2661,E1 10.4943,E2 474.6719} C_DIS
LIN {X 123.2349,Y -63.8527,Z 167,A -26.3438,B 10.3457,C 0.2757,E1 10.4909,E2 477.4559} C_DIS
LIN {X 121.1025,Y -67.8102,Z 167,A -28.1532,B 10.3457,C 0.2794,E1 10.4885,E2 479.2614} C_DIS
LIN {X 119.6412,Y -70.3562,Z 167,A -29.3443,B 10.3456,C 0.282,E1 10.4868,E2 480.4512} C_DIS
LIN {X 117.173,Y -74.395,Z 167,A -31.2708,B 10.3454,C 0.2862,E1 10.4839,E2 482.3763} C_DIS
LIN {X 112.9669,Y -80.638,Z 167,A -34.5659,B 10.3451,C 0.2987,E1 10.4787,E2 485.6988} C_DIS
LIN {X 110.9304,Y -83.4176,Z 167,A -35.7732,B 10.3451,C 0.2966,E1 10.4767,E2 486.8801} C_DIS
LIN {X 108.2036,Y -86.9256,Z 167,A -37.5385,B 10.3451,C 0.2992,E1 10.4737,E2 488.6387} C_DIS
LIN {X 105.3899,Y -90.3166,Z 167,A -39.4081,B 10.3449,C 0.3047,E1 10.4703,E2 490.5167} C_DIS
LIN {X 102.1239,Y -93.9932,Z 167,A -41.3727,B 10.3449,C 0.3076,E1 10.4666,E2 492.475} C_DIS
LIN {X 98.8894,Y -97.3907,Z 167,A -43.0541,B 10.3449,C 0.3054,E1 10.4634,E2 494.1257} C_DIS
LIN {X 97.1622,Y -99.1136,Z 167,A -44.2616,B 10.3447,C 0.3126,E1 10.461,E2 495.36} C_DIS
LIN {X 93.6549,Y -102.4348,Z 167,A -46.5087,B 10.3444,C 0.3231,E1 10.4563,E2 497.6416} C_DIS
LIN {X 90.9603,Y -104.835,Z 167,A -47.7376,B 10.3444,C 0.3196,E1 10.4538,E2 498.8386} C_DIS
LIN {X 88.2321,Y -107.1412,Z 167,A -49.2307,B 10.3444,C 0.323,E1 10.4506,E2 500.3356} C_DIS
LIN {X 84.7475,Y -109.9181,Z 167,A -51.0945,B 10.3442,C 0.3271,E1 10.4465,E2 502.2044} C_DIS
LIN {X 80.1155,Y -113.3381,Z 167,A -53.3909,B 10.3442,C 0.3294,E1 10.4413,E2 504.4927} C_DIS
LIN {X 76.276,Y -115.9568,Z 167,A -55.076,B 10.3442,C 0.3269,E1 10.4374,E2 506.1497} C_DIS
LIN {X 71.1321,Y -119.1815,Z 167,A -57.7581,B 10.344,C 0.3354,E1 10.431,E2 508.8568} C_DIS
LIN {X 67.2067,Y -121.4383,Z 167,A -59.6087,B 10.344,C 0.3378,E1 10.4265,E2 510.7067} C_DIS
LIN {X 63.4813,Y -123.4257,Z 167,A -61.1524,B 10.344,C 0.3355,E1 10.4228,E2 512.2263} C_DIS
LIN {X 57.9905,Y -126.0977,Z 167,A -63.8012,B 10.3438,C 0.3421,E1 10.4161,E2 514.8938} C_DIS
LIN {X 53.8678,Y -127.9136,Z 167,A -65.6539,B 10.3437,C 0.3443,E1 10.4113,E2 516.7472} C_DIS
LIN {X 50.4966,Y -129.2811,Z 167,A -67.1446,B 10.3437,C 0.3458,E1 10.4074,E2 518.2376} C_DIS
LIN {X 46.5031,Y -130.772,Z 167,A -68.8708,B 10.3437,C 0.347,E1 10.4029,E2 519.961} C_DIS
LIN {X 42.4817,Y -132.132,Z 167,A -70.6038,B 10.3436,C 0.3484,E1 10.3983,E2 521.6928} C_DIS
LIN {X 39.2394,Y -133.1309,Z 167,A -72.0654,B 10.3435,C 0.3512,E1 10.3944,E2 523.1633} C_DIS
LIN {X 35.6155,Y -134.1457,Z 167,A -73.4836,B 10.3435,C 0.3493,E1 10.3906,E2 524.5652} C_DIS
LIN {X 32.7085,Y -134.884,Z 167,A -74.8018,B 10.3435,C 0.3523,E1 10.387,E2 525.8946} C_DIS
LIN {X 29.1203,Y -135.7039,Z 167,A -77.2756,B 10.3426,C 0.3759,E1 10.3799,E2 528.4908} C_DIS
LIN {X 21.9965,Y -137.0412,Z 167,A -79.2311,B 10.3434,C 0.3535,E1 10.3749,E2 530.3164} C_DIS
LIN {X 15.598,Y -137.916,Z 167,A -82.0874,B 10.3432,C 0.3593,E1 10.3669,E2 533.1989} C_DIS
LIN {X 9.0958,Y -138.4961,Z 167,A -84.5451,B 10.3433,C 0.3547,E1 10.3602,E2 535.6277} C_DIS
LIN {X 5.8904,Y -138.6691,Z 167,A -86.0199,B 10.3433,C 0.3586,E1 10.356,E2 537.1224} C_DIS
LIN {X 2.8407,Y -138.7654,Z 167,A -87.4774,B 10.343,C 0.3634,E1 10.3518,E2 538.6059} C_DIS
LIN {X 2.8407,Y -138.7654,Z 167,A -87.4774,B 10.343,C 0.3634,E1 10.3518,E2 538.6059} C_DIS
Enddeposition()
LIN {X 0.9907,Y -139.7056,Z 167,A -87.695,B 10.3434,C 0.3571,E1 10.3515,E2 538.7884} C_DIS
Startdeposition()
$VEL.CP = VEL_PRINT
LIN {X 4.6632,Y -139.6328,Z 167,A -85.8494,B 10.3437,C 0.3488,E1 10.3568,E2 536.8978} C_DIS
LIN {X 9.4422,Y -139.3913,Z 167,A -83.6856,B 10.3439,C 0.3435,E1 10.3629,E2 534.7066} C_DIS
LIN {X 15.1126,Y -138.8891,Z 167,A -81.4628,B 10.3439,C 0.3452,E1 10.369,E2 532.4971} C_DIS
LIN {X 20.0203,Y -138.2671,Z 167,A -79.4823,B 10.3439,C 0.3452,E1 10.3745,E2 530.5217} C_DIS
LIN {X 23.5833,Y -137.7052,Z 167,A -78.0581,B 10.3438,C 0.3457,E1 10.3784,E2 529.1038} C_DIS
LIN {X 26.4845,Y -137.1756,Z 167,A -76.7744,B 10.3438,C 0.3431,E1 10.3819,E2 527.8096} C_DIS
LIN {X 32.3366,Y -135.9155,Z 167,A -74.52,B 10.3438,C 0.3462,E1 10.388,E2 525.5798} C_DIS
LIN {X 36.159,Y -134.9483,Z 167,A -72.7332,B 10.344,C 0.3406,E1 10.3929,E2 523.7696} C_DIS
LIN {X 39.9801,Y -133.868,Z 167,A -71.1485,B 10.344,C 0.3402,E1 10.3971,E2 522.1895} C_DIS
LIN {X 42.6864,Y -133.0277,Z 167,A -70.0059,B 10.344,C 0.3395,E1 10.4002,E2 521.0485} C_DIS
LIN {X 46.5036,Y -131.744,Z 167,A -68.3309,B 10.344,C 0.3372,E1 10.4046,E2 519.3693} C_DIS
LIN {X 49.3913,Y -130.6872,Z 167,A -67.0958,B 10.3441,C 0.3364,E1 10.4078,E2 518.1365} C_DIS
LIN {X 52.4102,Y -129.5054,Z 167,A -65.6872,B 10.3442,C 0.3328,E1 10.4115,E2 516.7164} C_DIS
LIN {X 55.8406,Y -128.0643,Z 167,A -64.1158,B 10.3443,C 0.3297,E1 10.4156,E2 515.1378} C_DIS
LIN {X 61.191,Y -125.5968,Z 167,A -61.8977,B 10.3443,C 0.3314,E1 10.4211,E2 512.9437} C_DIS
LIN {X 63.7271,Y -124.3279,Z 167,A -60.6331,B 10.3443,C 0.3272,E1 10.4243,E2 511.6647} C_DIS
LIN {X 67.3501,Y -122.4055,Z 167,A -58.9596,B 10.3445,C 0.3249,E1 10.4284,E2 509.9909} C_DIS
LIN {X 71.0221,Y -120.3118,Z 167,A -57.2514,B 10.3445,C 0.3228,E1 10.4325,E2 508.2844} C_DIS
LIN {X 75.2232,Y -117.7305,Z 167,A -55.223,B 10.3446,C 0.3193,E1 10.4374,E2 506.2533} C_DIS
LIN {X 78.8743,Y -115.3164,Z 167,A -53.3887,B 10.3448,C 0.3152,E1 10.4416,E2 504.4121} C_DIS
LIN {X 85.6954,Y -110.3418,Z 167,A -50.2563,B 10.3448,C 0.3172,E1 10.4486,E2 501.3197} C_DIS
LIN {X 88.3881,Y -108.1967,Z 167,A -48.6047,B 10.345,C 0.3084,E1 10.4522,E2 499.6354} C_DIS
Enddeposition()
END
